	    "DB_Alarme".MLD[18].%X0 := "Ventil_Stati_DB".Mld."SF_CM05.QM61";
	    "DB_Alarme".MLD[18].%X1 := "Ventil_Stati_DB".Mld."TO_auf_CM05.QM64";
	    "DB_Alarme".MLD[18].%X2 := "Ventil_Stati_DB".Mld."TO_zu_CM05.QM64";
	    "DB_Alarme".MLD[18].%X3 := "Ventil_Stati_DB".Mld."SF_CM05.QM64";
	    "DB_Alarme".MLD[18].%X4 := "Ventil_Stati_DB".Mld."TO_auf_GP01.QM15";
	    "DB_Alarme".MLD[18].%X5 := "Ventil_Stati_DB".Mld."TO_zu_GP01.QM15";
	    "DB_Alarme".MLD[18].%X6 := "Ventil_Stati_DB".Mld."SF_GP01.QM15";
	    "DB_Alarme".MLD[18].%X7 := "Ventil_Stati_DB".Mld."TO_auf_GP01.QM16";
	    "DB_Alarme".MLD[18].%X8 := "Ventil_Stati_DB".Mld."TO_zu_GP01.QM16";
	    "DB_Alarme".MLD[18].%X9 := "Ventil_Stati_DB".Mld."SF_GP01.QM16";
	    "DB_Alarme".MLD[18].%X10 := "Ventil_Stati_DB".Mld."TO_auf_GP01.QM17";
	    "DB_Alarme".MLD[18].%X11 := "Ventil_Stati_DB".Mld."TO_zu_GP01.QM17";
	    "DB_Alarme".MLD[18].%X12 := "Ventil_Stati_DB".Mld."SF_GP01.QM17";
	    "DB_Alarme".MLD[18].%X13 := "Ventil_Stati_DB".Mld."TO_auf_GP01.QM18";
	    "DB_Alarme".MLD[18].%X14 := "Ventil_Stati_DB".Mld."TO_zu_GP01.QM18";
	    "DB_Alarme".MLD[18].%X15 := "Ventil_Stati_DB".Mld."SF_GP01.QM18";
	    
	    "DB_Alarme".MLD[19].%X0 := "Ventil_Stati_DB".Mld."TO_auf_GP01.QM19";
	    "DB_Alarme".MLD[19].%X1 := "Ventil_Stati_DB".Mld."TO_zu_GP01.QM19";
	    "DB_Alarme".MLD[19].%X2 := "Ventil_Stati_DB".Mld."SF_GP01.QM19";
	    "DB_Alarme".MLD[19].%X3 := "Ventil_Stati_DB".Mld."TO_auf_GP01.QM20";
	    "DB_Alarme".MLD[19].%X4 := "Ventil_Stati_DB".Mld."TO_zu_GP01.QM20";
	    "DB_Alarme".MLD[19].%X5 := "Ventil_Stati_DB".Mld."SF_GP01.QM20";
	    "DB_Alarme".MLD[19].%X6 := "Ventil_Stati_DB".Mld."TO_auf_GP01.QM21";
	    "DB_Alarme".MLD[19].%X7 := "Ventil_Stati_DB".Mld."TO_zu_GP01.QM21";
	    "DB_Alarme".MLD[19].%X8 := "Ventil_Stati_DB".Mld."SF_GP01.QM21";
	    "DB_Alarme".MLD[19].%X9 := "Ventil_Stati_DB".Mld."TO_auf_GP01.QM22";
	    "DB_Alarme".MLD[19].%X10 := "Ventil_Stati_DB".Mld."TO_zu_GP01.QM22";
	    "DB_Alarme".MLD[19].%X11 := "Ventil_Stati_DB".Mld."SF_GP01.QM22";
	    "DB_Alarme".MLD[19].%X12 := "Ventil_Stati_DB".Mld."TO_auf_GP02.QM38";
	    "DB_Alarme".MLD[19].%X13 := "Ventil_Stati_DB".Mld."TO_zu_GP02.QM38";
	    "DB_Alarme".MLD[19].%X14 := "Ventil_Stati_DB".Mld."SF_GP02.QM38";
	    "DB_Alarme".MLD[19].%X15 := "Ventil_Stati_DB".Mld."TO_auf_GP02.QM39";
	    
	    "DB_Alarme".MLD[20].%X0 := "Ventil_Stati_DB".Mld."TO_zu_GP02.QM39";
	    "DB_Alarme".MLD[20].%X1 := "Ventil_Stati_DB".Mld."SF_GP02.QM39";
	    "DB_Alarme".MLD[20].%X2 := "Ventil_Stati_DB".Mld."TO_auf_GP02.QM40";
	    "DB_Alarme".MLD[20].%X3 := "Ventil_Stati_DB".Mld."TO_zu_GP02.QM40";
	    "DB_Alarme".MLD[20].%X4 := "Ventil_Stati_DB".Mld."SF_GP02.QM40";
	    "DB_Alarme".MLD[20].%X5 := "Ventil_Stati_DB".Mld."TO_auf_GP02.QM41";
	    "DB_Alarme".MLD[20].%X6 := "Ventil_Stati_DB".Mld."TO_zu_GP02.QM41";
	    "DB_Alarme".MLD[20].%X7 := "Ventil_Stati_DB".Mld."SF_GP02.QM41";
	    "DB_Alarme".MLD[20].%X8 := "Ventil_Stati_DB".Mld."TO_auf_GP02.QM42";
	    "DB_Alarme".MLD[20].%X9 := "Ventil_Stati_DB".Mld."TO_zu_GP02.QM42";
	    "DB_Alarme".MLD[20].%X10 := "Ventil_Stati_DB".Mld."SF_GP02.QM42";
	    "DB_Alarme".MLD[20].%X11 := "Ventil_Stati_DB".Mld."TO_auf_GP02.QM43";
	    "DB_Alarme".MLD[20].%X12 := "Ventil_Stati_DB".Mld."TO_zu_GP02.QM43";
	    "DB_Alarme".MLD[20].%X13 := "Ventil_Stati_DB".Mld."SF_GP02.QM43";
	    "DB_Alarme".MLD[20].%X14 := "Ventil_Stati_DB".Mld."TO_auf_GP02.QM44";
	    "DB_Alarme".MLD[20].%X15 := "Ventil_Stati_DB".Mld."TO_zu_GP02.QM44";
	    
	    "DB_Alarme".MLD[21].%X0 := "Ventil_Stati_DB".Mld."SF_GP02.QM44";
	    "DB_Alarme".MLD[21].%X1 := "Ventil_Stati_DB".Mld."TO_auf_GP02.QM45";
	    "DB_Alarme".MLD[21].%X2 := "Ventil_Stati_DB".Mld."TO_zu_GP02.QM45";
	    "DB_Alarme".MLD[21].%X3 := "Ventil_Stati_DB".Mld."SF_GP02.QM45";
	    "DB_Alarme".MLD[21].%X4 := "Ventil_Stati_DB".Mld."TO_auf_GP02.QM46";
	    "DB_Alarme".MLD[21].%X5 := "Ventil_Stati_DB".Mld."TO_zu_GP02.QM46";
	    "DB_Alarme".MLD[21].%X6 := "Ventil_Stati_DB".Mld."SF_GP02.QM46";
	    "DB_Alarme".MLD[21].%X7 := "Ventil_Stati_DB".Mld."TO_auf_GP01.QM14";
	    "DB_Alarme".MLD[21].%X8 := "Ventil_Stati_DB".Mld."TO_zu_GP01.QM14";
	    "DB_Alarme".MLD[21].%X9 := "Ventil_Stati_DB".Mld."SF_GP01.QM14";
	    "DB_Alarme".MLD[21].%X10 := "FP_CM01.GP01".Mld.Drucktest_Filter_ok;
	    "DB_Alarme".MLD[21].%X11 := "FP_CM01.GP01".Mld.Drucktest_Filter_Fehler;
	    "DB_Alarme".MLD[21].%X12 := "FP_CM02.GP04".Mld.Drucktest_Filter_ok;
	    "DB_Alarme".MLD[21].%X13 := "FP_CM02.GP04".Mld.Drucktest_Filter_Fehler;
	    "DB_Alarme".MLD[21].%X14 := "FP_CM01.GP01".Mld.Drucktest_Filter_erfordert;
	    "DB_Alarme".MLD[21].%X15 := "FP_CM02.GP04".Mld.Drucktest_Filter_erfordert;
	    
	    "DB_Alarme".MLD[22].%X0 := "DI_FW_1".MLD.Alarm_HW.PosSys;
	    "DB_Alarme".MLD[22].%X1 := "DI_FW_1".MLD.Alarm_HW.BE_rck;
	    "DB_Alarme".MLD[22].%X2 := "DI_FW_1".MLD.Alarm_HW.BE_vor;
	    "DB_Alarme".MLD[22].%X3 := "DI_FW_1".MLD.Alarm_HW.HubSys_li;
	    "DB_Alarme".MLD[22].%X4 := "DI_FW_1".MLD.Alarm_HW.HubSys_re;
	    "DB_Alarme".MLD[22].%X5 := "DI_FW_1".MLD.Alarm_HW.GE_oben_li;
	    "DB_Alarme".MLD[22].%X6 := "DI_FW_1".MLD.Alarm_HW.GE_unten_li;
	    "DB_Alarme".MLD[22].%X7 := "DI_FW_1".MLD.Alarm_HW.GE_oben_re;
	    "DB_Alarme".MLD[22].%X8 := "DI_FW_1".MLD.Alarm_HW.GE_unten_re;
	    "DB_Alarme".MLD[22].%X9 := "DI_FW_1".MLD.Alarm_HW.Koll_LF;
	    "DB_Alarme".MLD[22].%X10 := "DI_FW_1".MLD.Alarm_HW.Koll_WF;
	    "DB_Alarme".MLD[22].%X11 := "DI_FW_1".MLD.Alarm_HW.Afs_BS;
	    "DB_Alarme".MLD[22].%X12 := "DI_FW_1".MLD.Alarm_HW.Afs_WS;
	    "DB_Alarme".MLD[22].%X13 := "DI_FW_1".MLD.Alarm_HW.GurtUeL_li;
	    "DB_Alarme".MLD[22].%X14 := "DI_FW_1".MLD.Alarm_HW.GurtUeL_re;
	    "DB_Alarme".MLD[22].%X15 := "DI_FW_1".MLD.Alarm_HW.St_FU_Fahrt;
	    
	    "DB_Alarme".MLD[23].%X0 := "DI_FW_1".MLD.Alarm_HW.F_Brk_Hub_li;
	    "DB_Alarme".MLD[23].%X1 := "DI_FW_1".MLD.Alarm_HW.F_Brk_Hub_re;
	    "DB_Alarme".MLD[23].%X2 := "DI_FW_1".MLD.Alarm_HW.F_Brk_Fahr;
	    "DB_Alarme".MLD[23].%X3 := "DI_FW_1".MLD.Alarm_HW.St_FU_Hub_li;
	    "DB_Alarme".MLD[23].%X4 := "DI_FW_1".MLD.Alarm_HW.St_FU_Hub_re;
	    "DB_Alarme".MLD[23].%X5 := "DI_FW_1".MLD.Alarm_HW.Last_UeW_li;
	    "DB_Alarme".MLD[23].%X6 := "DI_FW_1".MLD.Alarm_HW.Last_UeW_re;
	    "DB_Alarme".MLD[23].%X7 := "DI_FW_1".MLD.Alarm_HW.Temp_Fahrt;
	    "DB_Alarme".MLD[23].%X8 := "DI_FW_1".MLD.Alarm_HW.Temp_Hub;
	    "DB_Alarme".MLD[23].%X9 := "DI_FW_1".MLD.Alarm_HW.Laser_TF;
	    "DB_Alarme".MLD[23].%X10 := "DI_FW_1".MLD.Alarm_HW.Laser_PL;
	    "DB_Alarme".MLD[23].%X11 := "DI_FW_1".MLD.Alarm_HW.Profinet_nok;
	    "DB_Alarme".MLD[23].%X12 := "DI_FW_1".MLD.Alarm_HW.res_1;
	    "DB_Alarme".MLD[23].%X13 := "DI_FW_1".MLD.Alarm_HW.res_2;
	    "DB_Alarme".MLD[23].%X14 := "DI_FW_1".MLD.Alarm_HW.res_3;
	    "DB_Alarme".MLD[23].%X15 := "DI_FW_1".MLD.Alarm_HW.res_4;
	    
	    "DB_Alarme".MLD[24].%X0 := "DI_FW_1".MLD.Alarm_SW.Fehler_Quitt;
	    "DB_Alarme".MLD[24].%X1 := "DI_FW_1".MLD.Alarm_SW.BA_ungueltig;
	    "DB_Alarme".MLD[24].%X2 := "DI_FW_1".MLD.Alarm_SW.ProgErr;
	    "DB_Alarme".MLD[24].%X3 := "DI_FW_1".MLD.Alarm_SW.nReferenz;
	    "DB_Alarme".MLD[24].%X4 := "DI_FW_1".MLD.Alarm_SW.NotStop;
	    "DB_Alarme".MLD[24].%X5 := "DI_FW_1".MLD.Alarm_SW.Laser_off;
	    "DB_Alarme".MLD[24].%X6 := "DI_FW_1".MLD.Alarm_SW.TO_Fahrt;
	    "DB_Alarme".MLD[24].%X7 := "DI_FW_1".MLD.Alarm_SW.Auto_SU;
	    "DB_Alarme".MLD[24].%X8 := "DI_FW_1".MLD.Alarm_SW.Auto_WT;
	    "DB_Alarme".MLD[24].%X9 := "DI_FW_1".MLD.Alarm_SW.WT_change;
	    "DB_Alarme".MLD[24].%X10 := "DI_FW_1".MLD.Alarm_SW.Hub_not_mittig_li;
	    "DB_Alarme".MLD[24].%X11 := "DI_FW_1".MLD.Alarm_SW.Hub_nen_li;
	    "DB_Alarme".MLD[24].%X12 := "DI_FW_1".MLD.Alarm_SW.TO_Hub_li;
	    "DB_Alarme".MLD[24].%X13 := "DI_FW_1".MLD.Alarm_SW.Senken_WT_li;
	    "DB_Alarme".MLD[24].%X14 := "DI_FW_1".MLD.Alarm_SW.Senken_Sperre_li;
	    "DB_Alarme".MLD[24].%X15 := "DI_FW_1".MLD.Alarm_SW.Heben_WT_li;
	    
	    "DB_Alarme".MLD[25].%X0 := "DI_FW_1".MLD.Alarm_SW.SO_fehlt_li;
	    "DB_Alarme".MLD[25].%X1 := "DI_FW_1".MLD.Alarm_SW.SU_fehlt_li;
	    "DB_Alarme".MLD[25].%X2 := "DI_FW_1".MLD.Alarm_SW.PosTyp_WT_Typ_li;
	    "DB_Alarme".MLD[25].%X3 := "DI_FW_1".MLD.Alarm_SW.WTon_bei_SU_li;
	    "DB_Alarme".MLD[25].%X4 := "DI_FW_1".MLD.Alarm_SW.TO_Hub_re;
	    "DB_Alarme".MLD[25].%X5 := "DI_FW_1".MLD.Alarm_SW.Senken_WT_re;
	    "DB_Alarme".MLD[25].%X6 := "DI_FW_1".MLD.Alarm_SW.Senken_Sperre_re;
	    "DB_Alarme".MLD[25].%X7 := "DI_FW_1".MLD.Alarm_SW.Heben_WT_re;
	    "DB_Alarme".MLD[25].%X8 := "DI_FW_1".MLD.Alarm_SW.SO_fehlt_re;
	    "DB_Alarme".MLD[25].%X9 := "DI_FW_1".MLD.Alarm_SW.SU_fehlt_re;
	    "DB_Alarme".MLD[25].%X10 := "DI_FW_1".MLD.Alarm_SW.PosTyp_WT_Typ_re;
	    "DB_Alarme".MLD[25].%X11 := "DI_FW_1".MLD.Alarm_SW.WTon_bei_SU_re;
	    "DB_Alarme".MLD[25].%X12 := "DI_FW_1".MLD.Alarm_SW.Hub_not_mittig_re;
	    "DB_Alarme".MLD[25].%X13 := "DI_FW_1".MLD.Alarm_SW.Hub_nen_re;
	    "DB_Alarme".MLD[25].%X14 := "DI_FW_1".MLD.Alarm_SW.ALSW_31;
	    "DB_Alarme".MLD[25].%X15 := "DI_FW_1".MLD.Alarm_SW.TO_Befehl;
	    
	    "DB_Alarme".MLD[26].%X0 := "DI_FW_1".MLD.Warnung.Optik_PosSys;
	    "DB_Alarme".MLD[26].%X1 := "DI_FW_1".MLD.Warnung.Temp_PosSys;
	    "DB_Alarme".MLD[26].%X2 := "DI_FW_1".MLD.Warnung.Temp_Fahrt;
	    "DB_Alarme".MLD[26].%X3 := "DI_FW_1".MLD.Warnung.Temp_Hub;
	    "DB_Alarme".MLD[26].%X4 := "DI_FW_1".MLD.Warnung.LSA;
	    "DB_Alarme".MLD[26].%X5 := "DI_FW_1".MLD.Warnung.Bh0;
	    "DB_Alarme".MLD[26].%X6 := "DI_FW_1".MLD.Warnung.Bh100;
	    "DB_Alarme".MLD[26].%X7 := "DI_FW_1".MLD.Warnung.Bh1000;
	    "DB_Alarme".MLD[26].%X8 := "DI_FW_1".MLD.Warnung.Wrn_Plaus_PosSys;
	    "DB_Alarme".MLD[26].%X9 := "DI_FW_1".MLD.Warnung.Wrn_WZ_niO_li_1;
	    "DB_Alarme".MLD[26].%X10 := "DI_FW_1".MLD.Warnung.Wrn_WZ_niO_li_2;
	    "DB_Alarme".MLD[26].%X11 := "DI_FW_1".MLD.Warnung.Wrn_WZ_niO_li_3;
	    "DB_Alarme".MLD[26].%X12 := "DI_FW_1".MLD.Warnung.Wrn_WZ_niO_li_4;
	    "DB_Alarme".MLD[26].%X13 := "DI_FW_1".MLD.Warnung.Wrn_WZ_niO_re_1;
	    "DB_Alarme".MLD[26].%X14 := "DI_FW_1".MLD.Warnung.Wrn_WZ_niO_re_2;
	    "DB_Alarme".MLD[26].%X15 := "DI_FW_1".MLD.Warnung.Wrn_WZ_niO_re_3;
	    
	    "DB_Alarme".MLD[27].%X0 := "DI_FW_1".MLD.Warnung.Wrn_WZ_niO_re_4;
	    "DB_Alarme".MLD[27].%X1 := "DI_FW_1".MLD.Warnung.WARN_18;
	    "DB_Alarme".MLD[27].%X2 := "DI_FW_1".MLD.Warnung.WARN_19;
	    "DB_Alarme".MLD[27].%X3 := "DI_FW_1".MLD.Warnung.WARN_20;
	    "DB_Alarme".MLD[27].%X4 := "DI_FW_1".MLD.Warnung.WARN_21;
	    "DB_Alarme".MLD[27].%X5 := "DI_FW_1".MLD.Warnung.WARN_22;
	    "DB_Alarme".MLD[27].%X6 := "DI_FW_1".MLD.Warnung.WARN_23;
	    "DB_Alarme".MLD[27].%X7 := "DI_FW_1".MLD.Warnung.WARN_24;
	    "DB_Alarme".MLD[27].%X8 := "DI_FW_1".MLD.Warnung.WARN_25;
	    "DB_Alarme".MLD[27].%X9 := "DI_FW_1".MLD.Warnung.WARN_26;
	    "DB_Alarme".MLD[27].%X10 := "DI_FW_1".MLD.Warnung.WARN_27;
	    "DB_Alarme".MLD[27].%X11 := "DI_FW_1".MLD.Warnung.WARN_28;
	    "DB_Alarme".MLD[27].%X12 := "DI_FW_1".MLD.Warnung.WARN_29;
	    "DB_Alarme".MLD[27].%X13 := "DI_FW_1".MLD.Warnung.WARN_30;
	    "DB_Alarme".MLD[27].%X14 := "DI_FW_1".MLD.Warnung.WARN_WT_nUms;
	    "DB_Alarme".MLD[27].%X15 := "DI_FW_1".MLD.Warnung.WARN_nAuto;
	    
	    "DB_Alarme".MLD[28].%X0 := "DI_QF_WR02_03".Mld.TO_WR02;
	    "DB_Alarme".MLD[28].%X1 := "DI_QF_WR02_03".Mld.TO_WR03;
	    "DB_Alarme".MLD[28].%X2 := "DI_QF_WR02_03".Mld.St_FU_WR02;
	    "DB_Alarme".MLD[28].%X3 := "DI_QF_WR02_03".Mld.St_FU_WR03;
	    "DB_Alarme".MLD[28].%X4 := "DI_QF_WR02_03".Mld.FU_nichtbereit_WR02;
	    "DB_Alarme".MLD[28].%X5 := "DI_QF_WR02_03".Mld.FU_nichtbereit_WR03;
	    "DB_Alarme".MLD[28].%X6 := "DI_QF_WR02_03".Mld.SF_WR02;
	    "DB_Alarme".MLD[28].%X7 := "DI_QF_WR02_03".Mld.SF_WR03;
	    "DB_Alarme".MLD[28].%X8 := FALSE;
	    "DB_Alarme".MLD[28].%X9 := "FP_CM01.GP01".Mld.Pu_Spuelen_Fertig;
	    "DB_Alarme".MLD[28].%X10 := "FP_CM02.GP04".Mld.Pu_Spuelen_Fertig;
	    "DB_Alarme".MLD[28].%X11 := "UP_CM01.GP02".Mld.Pu_Spuelen_Fertig;
	    "DB_Alarme".MLD[28].%X12 := "UP_CM02.GP05".Mld.Pu_Spuelen_Fertig;
	    "DB_Alarme".MLD[28].%X13 := "UP_CM03.GP03".Mld.Pu_Spuelen_Fertig;
	    "DB_Alarme".MLD[28].%X14 := "UP_CM04.GP06".Mld.Pu_Spuelen_Fertig;
	    "DB_Alarme".MLD[28].%X15 := "Pu_CM05.GP11_DB".Mld.Pu_Spuelen_Fertig;
	    
	    "DB_Alarme".MLD[29].%X0 := "DB_Korbumlaeufe".Korb[1].Warnung;
	    "DB_Alarme".MLD[29].%X1 := "DB_Korbumlaeufe".Korb[1].max_erreicht;
	    "DB_Alarme".MLD[29].%X2 := "DB_Korbumlaeufe".Korb[2].Warnung;
	    "DB_Alarme".MLD[29].%X3 := "DB_Korbumlaeufe".Korb[2].max_erreicht;
	    "DB_Alarme".MLD[29].%X4 := "DB_Korbumlaeufe".Korb[3].Warnung;
	    "DB_Alarme".MLD[29].%X5 := "DB_Korbumlaeufe".Korb[3].max_erreicht;
	    "DB_Alarme".MLD[29].%X6 := "DB_Korbumlaeufe".Korb[4].Warnung;
	    "DB_Alarme".MLD[29].%X7 := "DB_Korbumlaeufe".Korb[4].max_erreicht;
	    "DB_Alarme".MLD[29].%X8 := "DB_Korbumlaeufe".Korb[5].Warnung;
	    "DB_Alarme".MLD[29].%X9 := "DB_Korbumlaeufe".Korb[5].max_erreicht;
	    "DB_Alarme".MLD[29].%X10 := "DB_Korbumlaeufe".Korb[6].Warnung;
	    "DB_Alarme".MLD[29].%X11 := "DB_Korbumlaeufe".Korb[6].max_erreicht;
	    "DB_Alarme".MLD[29].%X12 := "DB_Korbumlaeufe".Korb[7].Warnung;
	    "DB_Alarme".MLD[29].%X13 := "DB_Korbumlaeufe".Korb[7].max_erreicht;
	    "DB_Alarme".MLD[29].%X14 := "DB_Korbumlaeufe".Korb[8].Warnung;
	    "DB_Alarme".MLD[29].%X15 := "DB_Korbumlaeufe".Korb[8].max_erreicht;
	        
	    "DB_Alarme".MLD[30].%X0 := "DB_Korbumlaeufe".Korb[9].Warnung;
	    "DB_Alarme".MLD[30].%X1 := "DB_Korbumlaeufe".Korb[9].max_erreicht;
	    "DB_Alarme".MLD[30].%X2 := "DB_Korbumlaeufe".Korb[10].Warnung;
	    "DB_Alarme".MLD[30].%X3 := "DB_Korbumlaeufe".Korb[10].max_erreicht;
	    "DB_Alarme".MLD[30].%X4 := "DB_Korbumlaeufe".Korb[11].Warnung;
	    "DB_Alarme".MLD[30].%X5 := "DB_Korbumlaeufe".Korb[11].max_erreicht;
	    "DB_Alarme".MLD[30].%X6 := "DB_Korbumlaeufe".Korb[12].Warnung;
	    "DB_Alarme".MLD[30].%X7 := "DB_Korbumlaeufe".Korb[12].max_erreicht;
	    "DB_Alarme".MLD[30].%X8 := "DB_Korbumlaeufe".Korb[13].Warnung;
	    "DB_Alarme".MLD[30].%X9 := "DB_Korbumlaeufe".Korb[13].max_erreicht;
	    "DB_Alarme".MLD[30].%X10 := "FP_CM01.GP01".Mld.Filterbeutel_Wechsel_Vorwarngrenze;
	    "DB_Alarme".MLD[30].%X11 := "FP_CM01.GP01".Mld.Filterbeutel_Wechsel_notwendig;
	    "DB_Alarme".MLD[30].%X12 := "FP_CM02.GP04".Mld.Filterbeutel_Wechsel_Vorwarngrenze;
	    "DB_Alarme".MLD[30].%X13 := "FP_CM02.GP04".Mld.Filterbeutel_Wechsel_notwendig;
	    "DB_Alarme".MLD[30].%X14 :=  "Pu_GP01.GP13".Mld.UeW_Dfl_Dos;
	    "DB_Alarme".MLD[30].%X15 := "Pu_GP02.GP10".Mld.UeW_Dfl_Dos;
	    
	    "DB_Alarme".MLD[31].%X0 := "FP_CM01.GP01".Mld.Drucktest_Pumpe_ok;
	    "DB_Alarme".MLD[31].%X1 := "FP_CM01.GP01".Mld.Drucktest_Pumpe_Fehler;
	    "DB_Alarme".MLD[31].%X2 := "FP_CM02.GP04".Mld.Drucktest_Pumpe_ok;
	    "DB_Alarme".MLD[31].%X3 := "FP_CM02.GP04".Mld.Drucktest_Pumpe_Fehler;
	    "DB_Alarme".MLD[31].%X4 := "UP_CM01.GP02".Mld.Drucktest_ok;
	    "DB_Alarme".MLD[31].%X5 := "UP_CM01.GP02".Mld.DT_Fehler;
	    "DB_Alarme".MLD[31].%X6 := "UP_CM02.GP05".Mld.Drucktest_ok;
	    "DB_Alarme".MLD[31].%X7 := "UP_CM02.GP05".Mld.DT_Fehler;
	    "DB_Alarme".MLD[31].%X8 := "UP_CM03.GP03".Mld.Drucktest_ok;
	    "DB_Alarme".MLD[31].%X9 := "UP_CM03.GP03".Mld.DT_Fehler;
	    "DB_Alarme".MLD[31].%X10 := "UP_CM04.GP06".Mld.Drucktest_ok;
	    "DB_Alarme".MLD[31].%X11 := "UP_CM04.GP06".Mld.DT_Fehler;
	    "DB_Alarme".MLD[31].%X12 := "Pu_CM05.GP11_DB".Mld.Drucktest_ok;
	    "DB_Alarme".MLD[31].%X13 := "Pu_CM05.GP11_DB".Mld.DT_Fehler;
	    "DB_Alarme".MLD[31].%X14 := "UP_CM01.GP02".Mld.UeW_Dfl_Ents;
	    "DB_Alarme".MLD[31].%X15 := "UP_CM02.GP05".Mld.UeW_Dfl_Ents;
	    
	        REGION Reserve
	        
	        "DB_Alarme".MLD[32].%X0 := FALSE;
	        "DB_Alarme".MLD[32].%X1 := FALSE;
	        "DB_Alarme".MLD[32].%X2 := FALSE;
	        "DB_Alarme".MLD[32].%X3 := FALSE;
	        "DB_Alarme".MLD[32].%X4 := FALSE;
	        "DB_Alarme".MLD[32].%X5 := FALSE;
	        "DB_Alarme".MLD[32].%X6 := FALSE;
	        "DB_Alarme".MLD[32].%X7 := FALSE;
	        "DB_Alarme".MLD[32].%X8 := FALSE;
	        "DB_Alarme".MLD[32].%X9 := FALSE;
	        "DB_Alarme".MLD[32].%X10 := FALSE;
	        "DB_Alarme".MLD[32].%X11 := FALSE;
	        "DB_Alarme".MLD[32].%X12 := FALSE;
	        "DB_Alarme".MLD[32].%X13 := FALSE;
	        "DB_Alarme".MLD[32].%X14 := FALSE;
	        "DB_Alarme".MLD[32].%X15 := FALSE;
	        
	        "DB_Alarme".MLD[33].%X0 := FALSE;
	        "DB_Alarme".MLD[33].%X1 := FALSE;
	        "DB_Alarme".MLD[33].%X2 := FALSE;
	        "DB_Alarme".MLD[33].%X3 := FALSE;
	        "DB_Alarme".MLD[33].%X4 := FALSE;
	        "DB_Alarme".MLD[33].%X5 := FALSE;
	        "DB_Alarme".MLD[33].%X6 := FALSE;
	        "DB_Alarme".MLD[33].%X7 := FALSE;
	        "DB_Alarme".MLD[33].%X8 := FALSE;
	        "DB_Alarme".MLD[33].%X9 := FALSE;
	        "DB_Alarme".MLD[33].%X10 := FALSE;
	        "DB_Alarme".MLD[33].%X11 := FALSE;
	        "DB_Alarme".MLD[33].%X12 := FALSE;
	        "DB_Alarme".MLD[33].%X13 := FALSE;
	        "DB_Alarme".MLD[33].%X14 := FALSE;
	        "DB_Alarme".MLD[33].%X15 := FALSE;
	        
	        "DB_Alarme".MLD[34].%X0 := FALSE;
	        "DB_Alarme".MLD[34].%X1 := FALSE;
	        "DB_Alarme".MLD[34].%X2 := FALSE;
	        "DB_Alarme".MLD[34].%X3 := FALSE;
	        "DB_Alarme".MLD[34].%X4 := FALSE;
	        "DB_Alarme".MLD[34].%X5 := FALSE;
	        "DB_Alarme".MLD[34].%X6 := FALSE;
	        "DB_Alarme".MLD[34].%X7 := FALSE;
	        "DB_Alarme".MLD[34].%X8 := FALSE;
	        "DB_Alarme".MLD[34].%X9 := FALSE;
	        "DB_Alarme".MLD[34].%X10 := FALSE;
	        "DB_Alarme".MLD[34].%X11 := FALSE;
	        "DB_Alarme".MLD[34].%X12 := FALSE;
	        "DB_Alarme".MLD[34].%X13 := FALSE;
	        "DB_Alarme".MLD[34].%X14 := FALSE;
	        "DB_Alarme".MLD[34].%X15 := FALSE;
	        
	        "DB_Alarme".MLD[35].%X0 := FALSE;
	        "DB_Alarme".MLD[35].%X1 := FALSE;
	        "DB_Alarme".MLD[35].%X2 := FALSE;
	        "DB_Alarme".MLD[35].%X3 := FALSE;
	        "DB_Alarme".MLD[35].%X4 := FALSE;
	        "DB_Alarme".MLD[35].%X5 := FALSE;
	        "DB_Alarme".MLD[35].%X6 := FALSE;
	        "DB_Alarme".MLD[35].%X7 := FALSE;
	        "DB_Alarme".MLD[35].%X8 := FALSE;
	        "DB_Alarme".MLD[35].%X9 := FALSE;
	        "DB_Alarme".MLD[35].%X10 := FALSE;
	        "DB_Alarme".MLD[35].%X11 := FALSE;
	        "DB_Alarme".MLD[35].%X12 := FALSE;
	        "DB_Alarme".MLD[35].%X13 := FALSE;
	        "DB_Alarme".MLD[35].%X14 := FALSE;
	        "DB_Alarme".MLD[35].%X15 := FALSE;
	        
	        "DB_Alarme".MLD[36].%X0 := FALSE;
	        "DB_Alarme".MLD[36].%X1 := FALSE;
	        "DB_Alarme".MLD[36].%X2 := FALSE;
	        "DB_Alarme".MLD[36].%X3 := FALSE;
	        "DB_Alarme".MLD[36].%X4 := FALSE;
	        "DB_Alarme".MLD[36].%X5 := FALSE;
	        "DB_Alarme".MLD[36].%X6 := FALSE;
	        "DB_Alarme".MLD[36].%X7 := FALSE;
	        "DB_Alarme".MLD[36].%X8 := FALSE;
	        "DB_Alarme".MLD[36].%X9 := FALSE;
	        "DB_Alarme".MLD[36].%X10 := FALSE;
	        "DB_Alarme".MLD[36].%X11 := FALSE;
	        "DB_Alarme".MLD[36].%X12 := FALSE;
	        "DB_Alarme".MLD[36].%X13 := FALSE;
	        "DB_Alarme".MLD[36].%X14 := FALSE;
	        "DB_Alarme".MLD[36].%X15 := FALSE;
	        
	        "DB_Alarme".MLD[37].%X0 := FALSE;
	        "DB_Alarme".MLD[37].%X1 := FALSE;
	        "DB_Alarme".MLD[37].%X2 := FALSE;
	        "DB_Alarme".MLD[37].%X3 := FALSE;
	        "DB_Alarme".MLD[37].%X4 := FALSE;
	        "DB_Alarme".MLD[37].%X5 := FALSE;
	        "DB_Alarme".MLD[37].%X6 := FALSE;
	        "DB_Alarme".MLD[37].%X7 := FALSE;
	        "DB_Alarme".MLD[37].%X8 := FALSE;
	        "DB_Alarme".MLD[37].%X9 := FALSE;
	        "DB_Alarme".MLD[37].%X10 := FALSE;
	        "DB_Alarme".MLD[37].%X11 := FALSE;
	        "DB_Alarme".MLD[37].%X12 := FALSE;
	        "DB_Alarme".MLD[37].%X13 := FALSE;
	        "DB_Alarme".MLD[37].%X14 := FALSE;
	        "DB_Alarme".MLD[37].%X15 := FALSE;
	        
	        "DB_Alarme".MLD[38].%X0 := FALSE;
	        "DB_Alarme".MLD[38].%X1 := FALSE;
	        "DB_Alarme".MLD[38].%X2 := FALSE;
	        "DB_Alarme".MLD[38].%X3 := FALSE;
	        "DB_Alarme".MLD[38].%X4 := FALSE;
	        "DB_Alarme".MLD[38].%X5 := FALSE;
	        "DB_Alarme".MLD[38].%X6 := FALSE;
	        "DB_Alarme".MLD[38].%X7 := FALSE;
	        "DB_Alarme".MLD[38].%X8 := FALSE;
	        "DB_Alarme".MLD[38].%X9 := FALSE;
	        "DB_Alarme".MLD[38].%X10 := FALSE;
	        "DB_Alarme".MLD[38].%X11 := FALSE;
	        "DB_Alarme".MLD[38].%X12 := FALSE;
	        "DB_Alarme".MLD[38].%X13 := FALSE;
	        "DB_Alarme".MLD[38].%X14 := FALSE;
	        "DB_Alarme".MLD[38].%X15 := FALSE;
	        
	        "DB_Alarme".MLD[39].%X0 := FALSE;
	        "DB_Alarme".MLD[39].%X1 := FALSE;
	        "DB_Alarme".MLD[39].%X2 := FALSE;
	        "DB_Alarme".MLD[39].%X3 := FALSE;
	        "DB_Alarme".MLD[39].%X4 := FALSE;
	        "DB_Alarme".MLD[39].%X5 := FALSE;
	        "DB_Alarme".MLD[39].%X6 := FALSE;
	        "DB_Alarme".MLD[39].%X7 := FALSE;
	        "DB_Alarme".MLD[39].%X8 := FALSE;
	        "DB_Alarme".MLD[39].%X9 := FALSE;
	        "DB_Alarme".MLD[39].%X10 := FALSE;
	        "DB_Alarme".MLD[39].%X11 := FALSE;
	        "DB_Alarme".MLD[39].%X12 := FALSE;
	        "DB_Alarme".MLD[39].%X13 := FALSE;
	        "DB_Alarme".MLD[39].%X14 := FALSE;
	        "DB_Alarme".MLD[39].%X15 := FALSE;
	        
	        "DB_Alarme".MLD[40].%X0 := FALSE;
	        "DB_Alarme".MLD[40].%X1 := FALSE;
	        "DB_Alarme".MLD[40].%X2 := FALSE;
	        "DB_Alarme".MLD[40].%X3 := FALSE;
	        "DB_Alarme".MLD[40].%X4 := FALSE;
	        "DB_Alarme".MLD[40].%X5 := FALSE;
	        "DB_Alarme".MLD[40].%X6 := FALSE;
	        "DB_Alarme".MLD[40].%X7 := FALSE;
	        "DB_Alarme".MLD[40].%X8 := FALSE;
	        "DB_Alarme".MLD[40].%X9 := FALSE;
	        "DB_Alarme".MLD[40].%X10 := FALSE;
	        "DB_Alarme".MLD[40].%X11 := FALSE;
	        "DB_Alarme".MLD[40].%X12 := FALSE;
	        "DB_Alarme".MLD[40].%X13 := FALSE;
	        "DB_Alarme".MLD[40].%X14 := FALSE;
	        "DB_Alarme".MLD[40].%X15 := FALSE;
	    END_REGION ;
	    
	END_REGION
	
	"FC_Mld_Leuchte_Hupe"(Max_Word := "Anzahl_Alarm_Woerter",
	                      La_Rot => #La_Rot,
	                      La_Gelb => #La_Gelb,
	                      La_Blau => #La_Blau);
	
	REGION Hupe
	    
	    //Quittung Hupe Rot
	    "DB_Alarme".Timer_Hupe_Rot.TON(IN := NOT "DB_Alarme".M_Q_Hupe_Rot AND NOT "DB_Alarme".Hupe_Dauer_Rot,
	    PT := "DB_Alarme".Zeit_Auto_Quitt_Hupe_Rot,
	    Q => #Hupe_Quitt_Rot);
	    
	    IF "DB_Alarme".IN_Quitt_Hupe OR #Hupe_Quitt_Rot THEN
	        "DB_Alarme".M_Q_Hupe_Rot := true;
	        "DB_Alarme".Hupe_Dauer_Rot := FALSE;
	    END_IF;
	    
	    //Quittung Hupe Gelb
	    "DB_Alarme".Timer_Hupe_Gelb.TON(IN := NOT "DB_Alarme".M_Q_Hupe_Gelb AND NOT "DB_Alarme".Hupe_Dauer_Gelb,
	    PT := "DB_Alarme".Zeit_Auto_Quitt_Hupe_Gelb,
	    Q => #Hupe_Quitt_Gelb);
	    
	    IF "DB_Alarme".IN_Quitt_Hupe OR #Hupe_Quitt_Gelb THEN
	        "DB_Alarme".M_Q_Hupe_Gelb := true;
	        "DB_Alarme".Hupe_Dauer_Gelb := FALSE;
	    END_IF;
	    
	    //Quittung Hupe Blau
	    "DB_Alarme".Timer_Hupe_Blau.TON(IN := NOT "DB_Alarme".M_Q_Hupe_Blau AND NOT "DB_Alarme".Hupe_Dauer_Blau,
	    PT := "DB_Alarme".Zeit_Auto_Quitt_Hupe_Blau,
	    Q => #Hupe_Quitt_Blau);
	    
	    IF "DB_Alarme".IN_Quitt_Hupe OR #Hupe_Quitt_Blau  THEN
	        "DB_Alarme".M_Q_Hupe_Blau := true;
	        "DB_Alarme".Hupe_Dauer_Blau := FALSE;
	    END_IF;
	    
	    //Ausgänge beschreiben
	    "DB_ANLAGE".OUT.Stoerung_Aku  := NOT "DB_Alarme".M_Q_Hupe_Rot;
	    "DB_Alarme".Lampe_Rot := #La_Rot;
	    "DB_Alarme".Lampe_Gelb := #La_Gelb;
	    "DB_Alarme".Lampe_Blau := #La_Blau;
	    
	    "DB_ANLAGE".OUT.Fehler_Quitt := "DI_FW_1".ZST.FEHLER OR NOT "DB_PNOZ_Comm".connection.activate
	    OR "Deckel_CM01".Zst.Fehler OR "Deckel_CM02".Zst.Fehler OR "Tor".Zst.Fehler
	    OR "DI_QF_WR02_03".Zst.Fehler OR "DB_Alarme".La_Quit_Err;
	    
	END_REGION
	
END_FUNCTION

FUNCTION "FC_Mld_Leuchte_Hupe" : Void
{ S7_Optimized_Access := 'TRUE' }
VERSION : 0.1
   VAR_INPUT 
      Max_Word : Int;   // Anzahl Worte insgesamt
   END_VAR

   VAR_OUTPUT 
      La_Rot : Bool;
      La_Gelb : Bool;
      La_Blau : Bool;
   END_VAR

   VAR_TEMP 
      i : Int;
      j : Int;
      Temp_Mld : Array[0..15] of Bool;   // Inhalt eines Meldewortes
      Temp_AM_Mld : Array[0..15] of Bool;   // Inhalt des Altmerkerwortes
      Edit_Mld_change : Bool;
   END_VAR


BEGIN
	REGION Parameter
	    //für Editierfunktion in Visu
	    //Meldenummer fängt in Visu bei 1 an, daher -1 für Wort und Bitberechnung
	    
	    //Adressberechnung
	    "DB_Alarme".Edit.Edit_Meldewort := ("DB_Alarme".Edit.Edit_Meld - 1) / 16; //welches Meldewort
	    "DB_Alarme".Edit.Edit_Meldebit := ("DB_Alarme".Edit.Edit_Meld - 1) MOD 16; //welches Meldebit
	    
	    //Änderung der ausgewählten Meldung in Visu erkannt
	    "FC_Flanke"(In:="DB_Alarme".Edit.Edit_Meld <> "DB_Alarme".Edit.Edit_Meld_old,
	                  neg:=FALSE,
	                  Flanke=>#Edit_Mld_change,
	                  AM:="DB_Alarme".Edit.AM_Edit);
	    
	    //Neue Daten in Editierstruktur
	    IF #Edit_Mld_change AND "DB_Alarme".Edit.Edit_Meld <> 0 THEN
	        "DB_Alarme".Edit.Par := "DB_Alarme".Para_Mld["DB_Alarme".Edit.Edit_Meldewort].Parameter["DB_Alarme".Edit.Edit_Meldebit];
	        
	        "DB_Alarme".Edit.Edit_Meld_old := "DB_Alarme".Edit.Edit_Meld; //Altmerker
	        "DB_Alarme".Edit.Uebernommen := FALSE;
	    END_IF;
	    
	    //Daten übernehmen
	    IF "DB_Alarme".Edit.Uebernehmen THEN
	        "DB_Alarme".Para_Mld["DB_Alarme".Edit.Edit_Meldewort].Parameter["DB_Alarme".Edit.Edit_Meldebit] := "DB_Alarme".Edit.Par;
	        "DB_Alarme".Edit.Uebernommen := TRUE;
	        "DB_Alarme".Edit.Uebernehmen := FALSE;
	    END_IF;
	    
	    // Cancel changes
	    IF "DB_Alarme".Edit.Verwerfen THEN
	        "DB_Alarme".Edit.Par := "DB_Alarme".Para_Mld["DB_Alarme".Edit.Edit_Meldewort].Parameter["DB_Alarme".Edit.Edit_Meldebit];
	        "DB_Alarme".Edit.Verwerfen := FALSE;
	    END_IF;
	    
	    "DB_Alarme".Edit.Editiert := "FC_Alarm_Editiert_HMI"(IN1:="DB_Alarme".Para_Mld["DB_Alarme".Edit.Edit_Meldewort].Parameter["DB_Alarme".Edit.Edit_Meldebit], IN2:="DB_Alarme".Edit.Par);
	        
	END_REGION
	
	REGION Auswertung
	    //Parameterbyte:
	    //Hupe Rot und Lampe Rot sind Standard, alles andere wird übers Parabyte eingestellt
	    //generell Hupe automatisch Quittieren pro Meldung, wenn Dauerhupen gewünscht dann im Parabyte einstellen
	    
	    //Init Meldeleuchten und Hupenquittung
	    #La_Rot := FALSE;
	    #La_Gelb := FALSE;
	    #La_Blau := FALSE;
	    "DB_Alarme".La_Quit_Err := FALSE;
	    "DB_Alarme".auto_aus := FALSE;
	    "DB_Alarme".stop_request := FALSE;
	    
	    FOR #i := 0 TO #Max_Word DO
	        
	        SCATTER(IN := "DB_Alarme".MLD[#i], //Meldewort in Bitarray vereinzeln
	                OUT => #Temp_Mld);
	        SCATTER(IN := "DB_Alarme".AM_MLD[#i], //Altmerkerwort in Bitarray vereinzeln
	                OUT => #Temp_AM_Mld);
	        
	        //Meldewort bearbeiten
	        FOR #j := 0 TO 15 DO
	            
	            //Lampen und sonstige Bits
	            IF #Temp_Mld[#j] = TRUE THEN
	                IF "DB_Alarme".Para_Mld[#i].Parameter[#j].La_Gelb = TRUE THEN
	                    #La_Gelb := TRUE;
	                END_IF;
	                
	                IF "DB_Alarme".Para_Mld[#i].Parameter[#j].La_Blau = TRUE THEN
	                    #La_Blau := TRUE;
	                END_IF;
	                
	                IF "DB_Alarme".Para_Mld[#i].Parameter[#j].nicht_La_Rot = FALSE THEN
	                    #La_Rot := TRUE;
	                END_IF;
	                
	                IF "DB_Alarme".Para_Mld[#i].Parameter[#j].La_Quit_Err = TRUE THEN
	                    "DB_Alarme".La_Quit_Err := TRUE;
	                END_IF;
	                
	            END_IF;
	            
	            //Hupen
	            IF ((#Temp_Mld[#j] XOR #Temp_AM_Mld[#j]) AND #Temp_Mld[#j]) = TRUE THEN
	                IF "DB_Alarme".Para_Mld[#i].Parameter[#j].Hupe_Gelb = TRUE THEN
	                    "DB_Alarme".M_Q_Hupe_Gelb := false;
	                    IF "DB_Alarme".Para_Mld[#i].Parameter[#j].Hupe_Dauer_Gelb = TRUE THEN
	                        "DB_Alarme".Hupe_Dauer_Gelb := TRUE;
	                    END_IF;
	                END_IF;
	                
	                IF "DB_Alarme".Para_Mld[#i].Parameter[#j].Hupe_Blau = TRUE THEN
	                    "DB_Alarme".M_Q_Hupe_Blau := false;
	                    IF "DB_Alarme".Para_Mld[#i].Parameter[#j].Hupe_Dauer_Blau = TRUE THEN
	                        "DB_Alarme".Hupe_Dauer_Blau := TRUE;
	                    END_IF;
	                END_IF;
	                
	                IF "DB_Alarme".Para_Mld[#i].Parameter[#j].nicht_Hupe_Rot = FALSE THEN
	                    "DB_Alarme".M_Q_Hupe_Rot := false;
	                    IF "DB_Alarme".Para_Mld[#i].Parameter[#j].Hupe_Dauer_Rot = TRUE THEN
	                        "DB_Alarme".Hupe_Dauer_Rot := TRUE;
	                    END_IF;
	                END_IF;
	            END_IF;
	            
	        END_FOR;
	        
	        //auf Altmerker kopieren
	        "DB_Alarme".AM_MLD[#i] := "DB_Alarme".MLD[#i];
	        
	    END_FOR;
	    
	END_REGION
END_FUNCTION

FUNCTION "FC_Flanke" : Void
{ S7_Optimized_Access := 'TRUE' }
VERSION : 0.1
   VAR_INPUT 
      In : Bool;
      neg : Bool;
   END_VAR

   VAR_OUTPUT 
      Flanke : Bool;
   END_VAR

   VAR_IN_OUT 
      AM : Bool;
   END_VAR


BEGIN
	IF (#In = TRUE AND #AM = FALSE AND #neg = FALSE) OR (#In = FALSE AND #AM = TRUE AND #neg = TRUE) THEN
	    #Flanke := TRUE;
	ELSE
	    #Flanke := false;
	END_IF;
	
	#AM := #In;
	
END_FUNCTION

FUNCTION "FC_Alarm_Editiert_HMI" : Bool
{ S7_Optimized_Access := 'TRUE' }
VERSION : 0.1
   VAR_INPUT 
      IN1 : "Alarm_Parameter";
      IN2 : "Alarm_Parameter";
   END_VAR


BEGIN
	#FC_Alarm_Editiert_HMI :=
	#IN1.Hupe_Blau       <> #IN2.Hupe_Blau OR
	#IN1.Hupe_Dauer_Blau <> #IN2.Hupe_Dauer_Blau OR
	#IN1.Hupe_Dauer_Gelb <> #IN2.Hupe_Dauer_Gelb OR
	#IN1.Hupe_Dauer_Rot  <> #IN2.Hupe_Dauer_Rot OR
	#IN1.Hupe_Gelb       <> #IN2.Hupe_Gelb OR
	#IN1.La_Blau         <> #IN2.La_Blau OR
	#IN1.La_Gelb         <> #IN2.La_Gelb OR
	#IN1.La_Quit_Err <> #IN2.La_Quit_Err OR
	#IN1.nicht_Hupe_Rot  <> #IN2.nicht_Hupe_Rot OR
	#IN1.nicht_La_Rot    <> #IN2.nicht_La_Rot;
END_FUNCTION

FUNCTION "FC_OUTPUT" : Void   // FC211, STL
TITLE = Schreiben der physikalischen Ausgänge
{ S7_Optimized_Access := 'FALSE' }
AUTHOR : RE
// stored: AutoNumber false
   VAR_TEMP
      Frg_Heben_li : Bool;
      Frg_Heben_re : Bool;
      Frg_Senken_li : Bool;
      Frg_Senken_re : Bool;
      Returnwert : Int;   // Rückgabewert SFC
      RetVal : Int;
   END_VAR
BEGIN

NETWORK
TITLE = Ausgabe
// Lampen

      A     "DB_ANLAGE".BA.Simulation;
      BEC;
//Warnung
      A     "DB_Alarme".Lampe_Gelb;
      O     "DB_ANLAGE".IN.Lamp_Test;
      =     "A_Mld_Wrn";
      =     "A_Mld_Wrn(2)";
      =     "A_Mld_Wrn_Geb.G";
// Störung
      A     "DB_Alarme".Lampe_Rot;
      O     "DB_ANLAGE".IN.Lamp_Test;
      =     "A_Mld_Al";
      =     "A_Mld_Al(2)";
      =     "A_Mld_Al_Geb.G";
//Hupe
      A     "DB_ANLAGE".OUT.Stoerung_Aku;
      =     "A_Hupe";
      =     "A_Hupe(2)";
      =     "A_Hupe_Geb.G";

//Fertigmeldung 1 WT will raus: CMD = 25
      L     "DB_WT1".akt_CMD;
      L     25;
      ==I;
      A     "DB_POS".POS["DB_WT1".POS].fertig;
      O(;
      L     "DB_WT2".akt_CMD;
      ==I;
      A     "DB_POS".POS["DB_WT2".POS].fertig;
      );
      O(;
      L     "DB_WT3".akt_CMD;
      L     25;
      ==I;
      A     "DB_POS".POS["DB_WT3".POS].fertig;
      );
      O(;
      L     "DB_WT4".akt_CMD;
      ==I;
      A     "DB_POS".POS["DB_WT4".POS].fertig;
      );
      O(;
      L     "DB_WT5".akt_CMD;
      L     25;
      ==I;
      A     "DB_POS".POS["DB_WT5".POS].fertig;
      );
      O(;
      L     "DB_WT6".akt_CMD;
      ==I;
      A     "DB_POS".POS["DB_WT6".POS].fertig;
      );
      O(;
      L     "DB_WT7".akt_CMD;
      L     25;
      ==I;
      A     "DB_POS".POS["DB_WT7".POS].fertig;
      );
      O(;
      L     "DB_WT8".akt_CMD;
      ==I;
      A     "DB_POS".POS["DB_WT8".POS].fertig;
      );
      O(;
      L     "DB_WT9".akt_CMD;
      L     25;
      ==I;
      A     "DB_POS".POS["DB_WT9".POS].fertig;
      );
      O(;
      L     "DB_WT10".akt_CMD;
      ==I;
      A     "DB_POS".POS["DB_WT10".POS].fertig;
      );
      O(;
      L     "DB_WT11".akt_CMD;
      L     25;
      ==I;
      A     "DB_POS".POS["DB_WT11".POS].fertig;
      );
      O(;
      L     "DB_WT12".akt_CMD;
      ==I;
      A     "DB_POS".POS["DB_WT12".POS].fertig;
      );
      A     "Clock_1Hz";
      O     "DI_FW_Auftrag_DB".Frg_Ausfahrt;
      O     "DB_ANLAGE".IN.Lamp_Test;
      =     "A_Mld_fertig";
      =     "A_Mld_fertig(2)";
      =     "A_Mld_fertig_Geb.G";

      A     "DB_ANLAGE".OUT.Fehler_Quitt;
      O     "DB_ANLAGE".IN.Lamp_Test;
      =     "A_LED_Q_Err";
      L     3;
      JC    LED;
      L     0;
LED:  T     "MobilePanel".Drucktaster_K2_LED;

      AN    "DB_PNOZ_IN_Out".In.PNOZ_OK;
      =     "A_LED_Q_NH";

// Meldung Automatik
      A     "DB_ANLAGE".OUT.MD_Auto;
      O     "DB_ANLAGE".IN.Lamp_Test;
      =     "A_Mld_Automatik";
      =     "A_Mld_Automatik(2)";
      =     "A_Mld_Automatik_Geb.G";

// Turmleuchte Tür
      AN    "E_Wrn_Gas_ok";
      =     "A_TL_T_Vorarlarm_Gas";
      =     "A_TL_T_Vorarlarm_Gas(2)";

      AN    "E_Al_Gas_ok";
      =     "A_TL_T_Hauptalarm_Gas";
      =     "A_TL_T_Hauptalarm_Gas(2)";

      AN    "E_Al_Gas_ok";
      =     "A_TL_T_Hupe";
      =     "A_TL_T_Hupe(2)";

// Koppelsignale
// --> AWA
      SET;
      =     "A_KS_in_Betrieb";
// --> Wäscher
      AN    "E_Niv_max_CM05.BL01";
      A     "E_Niv_Uel_CM05.BL12";
      =     "A_KS_CM05_nicht_Voll";

// Werkschutz
// 14x Leckage
      A     "FP_CM02.GP04".Mld.Leckage;
      O     "Pu_CL01.GP08".Mld.Leckage;
      O     "Pu_CL02.GP09".Mld.Leckage;
      O     "Pu_GP01.GP12".Mld.Leckage;
      O     "Pu_GP02.GP07".Mld.Leckage;
      O     "Pu_GP01.GP13".Mld.Leckage_Pumpe;
      O     "Pu_GP01.GP13".Mld.Leckage_PFA_Uebergang;
      O     "Pu_GP01.GP13".Mld.Leckage_Doppelrohr;
      O     "Pu_GP01.GP13".Mld.Leckage_Uml_Tunnel;
      O     "Pu_GP02.GP10".Mld.Leckage_Pumpe;
      O     "Pu_GP02.GP10".Mld.Leckage_PFA_Uebergang;
      ON    "E_LS_GP02.BL26";
      O     "Pu_GP02.GP10".Mld.Leckage_Doppelschlauch;
      ON    "E_LS_GP02.BL33";
      =     "A_Mld_WS_Leckage";
// 3x Überlauf
      A     "UP_CM01.GP02".Mld.Niv_Ueberlauf;
      O     "UP_CM02.GP05".Mld.Niv_Ueberlauf;
      O     "Pu_CM05.GP11_DB".Mld."Uel_CM05.BL05";
      =     "A_Mld_WS_Ueberlauf";

      A     "DB_Alarme".Lampe_Rot;
      =     "A_Mld_WS_SSt";

// LED Türen
      AN    "DB_PNOZ_IN_Out".In.Tuer_VS_ok;
      A     "Clock_1Hz";
      =     "A_LED_Tuer_VS";

      AN    "DB_PNOZ_IN_Out".In.Tuer_RS_ok;
      A     "Clock_1Hz";
      =     "A_LED_Tuer_RS";


NETWORK
TITLE = FW
// Transportsystem
// Reparaturbetrieb
      A     "DB_ANLAGE".IN.Reparatur;
      A     "DB_ANLAGE".IN.BA_Tipp;
      =     "A_RepB";

//--------------------------
//FW1
//--------------------------
// FU Fahrt: FU[10]

      CALL  "FB_FU_OUT_TW", "DI_FU_Fahrt"
      ( Req_High       := "DI_FW_1".OUT.VOR,
        Req_Low        := "DI_FW_1".OUT.RUECK,
        Reglersperre   := "FU_In_Out".FU[10].PA.Steuerwort.RegSp,
        Freigabe_Stopp := "FU_In_Out".FU[10].PA.Steuerwort.FrgStop,
        Freigabe_Halt  := "FU_In_Out".FU[10].PA.Steuerwort.FrgHalt,
        Break_ok       := "DI_FW_POS_1".IN.Break_on,
        SollSpeed      := "DI_FW_POS_1".OUT.SollSpeed,
        Ist_Speed      := "DI_FW_POS_1".IN.IstSpeed,
        PAW_Speed      := "FU_In_Out".FU[10].PA.Speed,
        PEW_Speed      := "FU_In_Out".FU[10].PE.Speed
      );

      A     "DI_FW_1".OUT.VOR;
      O     "DI_FW_1".OUT.RUECK;
      =     "A_Frg_FU_Fahrt";

// FU Hub links: FU[11]
      A     "DI_FW_1".OUT.HEBEN_li;
      =     "A_Heb_li";
      A     "DI_FW_1".OUT.SENKEN_li;
      =     "A_Snk_li";

      A     "DI_FW_1".OUT.HEBEN_li;
      A     "A_RepB";
      O     "E_Frg_Heb_li";
      =     #Frg_Heben_li;

      A     "DI_FW_1".OUT.SENKEN_li;
      A     "A_RepB";
      O     "E_Frg_Snk_li";
      =     #Frg_Senken_li;

      CALL  "FB_FU_OUT_TW", "DI_FU_Hub_links"
      ( Req_High       := #Frg_Heben_li,
        Req_Low        := #Frg_Senken_li,
        Reglersperre   := "FU_In_Out".FU[11].PA.Steuerwort.RegSp,
        Freigabe_Stopp := "FU_In_Out".FU[11].PA.Steuerwort.FrgStop,
        Freigabe_Halt  := "FU_In_Out".FU[11].PA.Steuerwort.FrgHalt,
        Break_ok       := "DI_FW_HUB_links".IN.Break_on,
        SollSpeed      := "DI_FW_HUB_links".OUT.SollSpeed,
        Ist_Speed      := "DI_FW_HUB_links".IN.IstSpeed,
        PAW_Speed      := "FU_In_Out".FU[11].PA.Speed,
        PEW_Speed      := "FU_In_Out".FU[11].PE.Speed
      );

      A     "DI_FW_1".OUT.HEBEN_li;
      O     "DI_FW_1".OUT.SENKEN_li;
      =     "A_Frg_FU_Hub_li";

      A     "DI_FW_1".ZST.Tipp;
      A     "DI_FW_1".ZST.BEREIT;
      A     "DI_FW_1".ZST.Unten_li;
      A     "T_ErrQuitt";
      =     "A_WZ_Tara_li_1";
      =     "A_WZ_Tara_li_2";
      =     "A_WZ_Tara_li_3";
      =     "A_WZ_Tara_li_4";

// FU Hub rechts: FU[12]
      A     "DI_FW_1".OUT.HEBEN_re;
      =     "A_Heb_re";
      A     "DI_FW_1".OUT.SENKEN_re;
      =     "A_Snk_re";

      A     "DI_FW_1".OUT.HEBEN_re;
      A     "A_RepB";
      O     "E_Frg_Heb_re";
      =     #Frg_Heben_re;

      A     "DI_FW_1".OUT.SENKEN_re;
      A     "A_RepB";
      O     "E_Frg_Snk_re";
      =     #Frg_Senken_re;

      CALL  "FB_FU_OUT_TW", "DI_FU_Hub_rechts"
      ( Req_High       := #Frg_Heben_re,
        Req_Low        := #Frg_Senken_re,
        Reglersperre   := "FU_In_Out".FU[12].PA.Steuerwort.RegSp,
        Freigabe_Stopp := "FU_In_Out".FU[12].PA.Steuerwort.FrgStop,
        Freigabe_Halt  := "FU_In_Out".FU[12].PA.Steuerwort.FrgHalt,
        Break_ok       := "DI_FW_HUB_rechts".IN.Break_on,
        SollSpeed      := "DI_FW_HUB_rechts".OUT.SollSpeed,
        Ist_Speed      := "DI_FW_HUB_rechts".IN.IstSpeed,
        PAW_Speed      := "FU_In_Out".FU[12].PA.Speed,
        PEW_Speed      := "FU_In_Out".FU[12].PE.Speed
      );

      A     "DI_FW_1".OUT.HEBEN_re;
      O     "DI_FW_1".OUT.SENKEN_re;
      =     "A_Frg_FU_Hub_re";


      A     "DI_FW_1".ZST.Tipp;
      A     "DI_FW_1".ZST.BEREIT;
      A     "DI_FW_1".ZST.Unten_re;
      A     "T_ErrQuitt";
      =     "A_WZ_Tara_re_1";
      =     "A_WZ_Tara_re_2";
      =     "A_WZ_Tara_re_3";
      =     "A_WZ_Tara_re_4";


NETWORK
TITLE = Be- und Entladestände (QF1 / QF2)
// WR02/03
// QF 1 FU[8]

      CALL  "FB_FU_OUT_TW", "DI_FU_WR02"
      ( Req_High       := "DI_QF_WR02_03".Out.WR02_einfahren,
        Req_Low        := "DI_QF_WR02_03".Out.WR02_ausfahren,
        Reglersperre   := "FU_In_Out".FU[8].PA.Steuerwort.RegSp,
        Freigabe_Stopp := "FU_In_Out".FU[8].PA.Steuerwort.FrgStop,
        Freigabe_Halt  := "FU_In_Out".FU[8].PA.Steuerwort.FrgHalt,
        Break_ok       := ,
        SollSpeed      := "DI_QF_WR02_03".Out.Soll_speed_WR02,
        Ist_Speed      := "DI_QF_WR02_03".In.FU_speed_WR02,
        PAW_Speed      := "FU_In_Out".FU[8].PA.Speed,
        PEW_Speed      := "FU_In_Out".FU[8].PE.Speed
      );

      A     "DI_QF_WR02_03".Out.WR02_einfahren;
      O     "DI_QF_WR02_03".Out.WR02_ausfahren;
      =     "A_Frg_FU_QF_WR02";

// QF 2 FU[9]

      CALL  "FB_FU_OUT_TW", "DI_FU_WR03"
      ( Req_High       := "DI_QF_WR02_03".Out.WR03_einfahren,
        Req_Low        := "DI_QF_WR02_03".Out.WR03_ausfahren,
        Reglersperre   := "FU_In_Out".FU[9].PA.Steuerwort.RegSp,
        Freigabe_Stopp := "FU_In_Out".FU[9].PA.Steuerwort.FrgStop,
        Freigabe_Halt  := "FU_In_Out".FU[9].PA.Steuerwort.FrgHalt,
        Break_ok       := ,
        SollSpeed      := "DI_QF_WR02_03".Out.Soll_speed_WR03,
        Ist_Speed      := "DI_QF_WR02_03".In.FU_speed_WR03,
        PAW_Speed      := "FU_In_Out".FU[9].PA.Speed,
        PEW_Speed      := "FU_In_Out".FU[9].PE.Speed
      );

      A     "DI_QF_WR02_03".Out.WR03_einfahren;
      O     "DI_QF_WR02_03".Out.WR03_ausfahren;
      =     "A_Frg_FU_QF_WR03";


NETWORK
TITLE = 
// Ausgänge
      CALL  "Output_Peripherie";

END_FUNCTION

FUNCTION_BLOCK "FB_FU_OUT_TW"   // FB12, LAD
TITLE = Ausgabe Einzel-FU
{ S7_Optimized_Access := 'TRUE' }
// stored: AutoNumber false, IsIECCheckEnabled true, MemoryReserve 100, SetENOAutomatically false
   VAR_INPUT
      Req_High : Bool;   // Anforderung Vorwärts/Heben
      Req_Low : Bool;   // Anforderun Rückwärts/Senken
   END_VAR
   VAR_IN_OUT
      Reglersperre : Bool;
      Freigabe_Stopp : Bool;
      Freigabe_Halt : Bool;
      Break_ok : Bool;
      SollSpeed : Int;   // Geschwindigkeit Fahren in %
      Ist_Speed : Int;
      PAW_Speed : Int;
      PEW_Speed : Int;
   END_VAR
   VAR RETAIN
      maxSpeed : Real := 7500.0;   // maximale Ausgabe (entspricht 100%)
      Faktor { ExternalAccessible := 'False'; ExternalVisible := 'False'; ExternalWritable := 'False'} : Real := 100.0;
      minSpeed : Int := 750;   // Freigabe nehmen unterhalb diesen Wertes im PEW
   END_VAR
   VAR_TEMP
      TempSpeed : Real;
      Faktor_Sim : Real;
      Delta : Int;
   END_VAR
BEGIN

REGION Network 1 (SCL): Istwert erfassen
   REGION Istwert erfassen
       // Statement section REGION
       #Ist_Speed:=REAL_TO_INT((INT_TO_REAL(#PEW_Speed)/#maxSpeed) * #Faktor);
   END_REGION
END_REGION

REGION Network 2 (SCL): Ausgabe Speed
   REGION Ausgabe Speed

       //Not-Halt --> sofort aus
       IF "DB_ANLAGE".BA.Not_Aus THEN
           #Reglersperre := TRUE;
           #Freigabe_Stopp := FALSE;
           #PAW_Speed := 0;

           //vorwärts/hoch positive Ausgabe    
       ELSIF #Req_High AND #SollSpeed <> 0 THEN
           #Reglersperre := FALSE;
           #Freigabe_Stopp := TRUE;
           #PAW_Speed := REAL_TO_INT(INT_TO_REAL(#SollSpeed) / #Faktor * #maxSpeed);

           //rückwärts/runter negative Ausgabe    
       ELSIF #Req_Low AND #SollSpeed <> 0 THEN
           #Reglersperre := FALSE;
           #Freigabe_Stopp := TRUE;
           #PAW_Speed := REAL_TO_INT(INT_TO_REAL(#SollSpeed) / #Faktor * #maxSpeed * -1.0);

           //sonst aus    
       ELSE
           #Freigabe_Stopp := #PEW_Speed >= #minSpeed;
           #Reglersperre := FALSE;
           #PAW_Speed := 0;
       END_IF;

       #Freigabe_Halt := #Freigabe_Stopp;
       #Break_ok := NOT #Freigabe_Stopp AND #Ist_Speed=0;

   END_REGION
END_REGION

REGION Network 3 (SCL): Simulation
   REGION Simulation

       IF "DB_ANLAGE".BA.Simulation THEN

           //Abfahrrampe berechnen
           #Faktor_Sim := 15.0; //500ms von 7500 auf 0 (7500.0/500.0)
           //Korrekturwert berechnen
           #Delta := REAL_TO_INT(#Faktor_Sim * INT_TO_REAL("DI_FW_MANAGER".akt_CT));

           //Geschwindigkeit reduzieren
           IF #PEW_Speed > #PAW_Speed THEN
               #PEW_Speed := #PEW_Speed - #Delta;
               IF #PEW_Speed <= #PAW_Speed THEN
                   #PEW_Speed := #PAW_Speed;
               END_IF;

               //Geschwindigkeit erhöhen
           ELSIF #PEW_Speed < #PAW_Speed THEN
               #PEW_Speed := #PEW_Speed + #Delta;
               IF #PEW_Speed >= #PAW_Speed THEN
                   #PEW_Speed := #PAW_Speed;
               END_IF;

           ELSE
               #PEW_Speed := #PAW_Speed;
           END_IF; 

       END_IF;
   END_REGION
END_REGION
END_FUNCTION_BLOCK

FUNCTION "Output_Peripherie" : Void   // FC1011, LAD
{ S7_Optimized_Access := 'TRUE' }
// stored: AutoNumber false, SetENOAutomatically true
BEGIN

REGION Network 1 (SCL): Schnellauftor
   "A_RT_auf" := "Tor".Out.auf;
   "A_RT_zu" := "Tor".Out.zu;
END_REGION

REGION Network 2 (SCL): Deckel
   // CM01
   "A_Dkl_li_auf_CM01" := "Deckel_CM01".Out.links_auf;
   "A_Dkl_li_zu_CM01" := "Deckel_CM01".Out.links_zu;
   "A_Dkl_re_auf_CM01" := "Deckel_CM01".Out.rechts_auf;
   "A_Dkl_re_zu_CM01" := "Deckel_CM01".Out.rechts_zu;
   // CM02
   "A_Dkl_li_auf_CM02" := "Deckel_CM02".Out.links_auf;
   "A_Dkl_li_zu_CM02" := "Deckel_CM02".Out.links_zu;
   "A_Dkl_re_auf_CM02" := "Deckel_CM02".Out.rechts_auf;
   "A_Dkl_re_zu_CM02" := "Deckel_CM02".Out.rechts_zu;
END_REGION

REGION Network 3 (SCL): CM01
   //Filtern
   // Pumpe (FU[1])
   "A_Frg_FU_FP_HQ01" := "FP_CM01.GP01".Out.GP0x_Ein;

   "FU_In_Out".FU[1].PA.Steuerwort.FrgHalt := "FP_CM01.GP01".Out.GP0x_Ein;
   "FU_In_Out".FU[1].PA.Steuerwort.FrgStop := "FP_CM01.GP01".Out.GP0x_Ein;
   "FU_In_Out".FU[1].PA.Steuerwort.RegSp := NOT "FU_In_Out".FU[1].PA.Steuerwort.FrgHalt;
   "FU_In_Out".FU[1].PA.Speed := "FP_CM01.GP01".Out.Soll_speed;

   // IF ("FP_CM01.GP01".In."Betriebsart" = 0) AND ("Panel".FP_CM01.BA = 1) THEN
   //     "Panel".FP_CM01.BA := 0; // Filtern
   // END_IF;

   //Ventile
   "A_CM01.QM18" := "FP_CM01.GP01".Out.Ventil_Saugseite;
   "A_CM01.QM19" := "FP_CM01.GP01".Out.Spülventil_P_Eingang;
   "A_HQ01.LV01" := "FP_CM01.GP01".Out.Ventil_Entlueften;
   "A_HQ01.QM21" := "FP_CM01.GP01".Out.Ventil_Eingang_Filter;
   "A_HQ01.QM22" := "FP_CM01.GP01".Out.Spülventil_F_Eingang;
   "A_HQ01.QM23" := "FP_CM01.GP01".Out.Ventil_Ausgang_Filter;
   "A_HQ01.QM24" := "FP_CM01.GP01".Out.Spülventil_Ausgang;

   // Umwälzen
   // Pumpe (FU[2])
   "A_Frg_FU_UP_HF_CM01" := "UP_CM01.GP02".Out.GP0x_Ein;

   "FU_In_Out".FU[2].PA.Steuerwort.FrgHalt := "UP_CM01.GP02".Out.GP0x_Ein;
   "FU_In_Out".FU[2].PA.Steuerwort.FrgStop := "UP_CM01.GP02".Out.GP0x_Ein;
   "FU_In_Out".FU[2].PA.Steuerwort.RegSp := NOT "FU_In_Out".FU[2].PA.Steuerwort.FrgHalt;
   "FU_In_Out".FU[2].PA.Speed := "UP_CM01.GP02".Out.Soll_speed;

   //Ventile
   "A_CM01.QM25" := "UP_CM01.GP02".Out.Ventil_Saugseite;
   "A_CM01.QM26" := "UP_CM01.GP02".Out.Ventil_Druckseite;
   "A_CM01.QM20" := "UP_CM01.GP02".Out.Spülventil_Eingang;
   "A_CM01.QM27" := "UP_CM01.GP02".Out.Spülventil_Ausgang;
   "A_GP02.QM45":= "UP_CM01.GP02".Out.Entsorgung_UV02;
   "A_GP02.QM44" := "UP_CM01.GP02".Out.Ventil_UV02_GP01 OR "UP_CM02.GP05".Out.Ventil_UV02_GP01;
   "A_GP02.QM43" := "UP_CM01.GP02".Out.Ventil_UV02_GP02 OR "UP_CM02.GP05".Out.Ventil_UV02_GP02;
END_REGION

REGION Network 4 (SCL): CM02
   //Filtern
   // Pumpe (FU[4])
   "A_Frg_FU_FP_HQ02" := "FP_CM02.GP04".Out.GP0x_Ein;

   "FU_In_Out".FU[4].PA.Steuerwort.FrgHalt := "FP_CM02.GP04".Out.GP0x_Ein;
   "FU_In_Out".FU[4].PA.Steuerwort.FrgStop := "FP_CM02.GP04".Out.GP0x_Ein;
   "FU_In_Out".FU[4].PA.Steuerwort.RegSp := NOT "FU_In_Out".FU[4].PA.Steuerwort.FrgHalt;
   "FU_In_Out".FU[4].PA.Speed := "FP_CM02.GP04".Out.Soll_speed;

   // IF ("FP_CM02.GP04".In."Betriebsart" = 0) AND ("Panel".FP_CM02.BA = 1) THEN
   //     "Panel".FP_CM02.BA := 0; // Filtern
   // END_IF;

   //Ventile
   "A_CM02.QM55" := "FP_CM02.GP04".Out.Ventil_Saugseite;
   "A_CM02.QM56" := "FP_CM02.GP04".Out.Spülventil_P_Eingang;
   "A_HQ02.LV02" := "FP_CM02.GP04".Out.Ventil_Entlueften;
   "A_HQ02.QM59" := "FP_CM02.GP04".Out.Ventil_Eingang_Filter;
   "A_HQ02.QM58" := "FP_CM02.GP04".Out.Spülventil_F_Eingang;
   "A_HQ02.QM60" := "FP_CM02.GP04".Out.Ventil_Ausgang_Filter;
   "A_HQ02.QM61" := "FP_CM02.GP04".Out.Spülventil_Ausgang;

   // Umwälzen
   // Pumpe (FU[5])
   "A_Frg_FU_UP_HF_CM02" := "UP_CM02.GP05".Out.GP0x_Ein;

   "FU_In_Out".FU[5].PA.Steuerwort.FrgHalt := "UP_CM02.GP05".Out.GP0x_Ein;
   "FU_In_Out".FU[5].PA.Steuerwort.FrgStop := "UP_CM02.GP05".Out.GP0x_Ein;
   "FU_In_Out".FU[5].PA.Steuerwort.RegSp := NOT "FU_In_Out".FU[5].PA.Steuerwort.FrgHalt;
   "FU_In_Out".FU[5].PA.Speed := "UP_CM02.GP05".Out.Soll_speed;

   //Ventile
   "A_CM02.QM62" := "UP_CM02.GP05".Out.Ventil_Saugseite;
   "A_CM02.QM63" := "UP_CM02.GP05".Out.Ventil_Druckseite;
   "A_CM02.QM57" := "UP_CM02.GP05".Out.Spülventil_Eingang;
   "A_CM02.QM64" := "UP_CM02.GP05".Out.Spülventil_Ausgang;
   "A_GP02.QM46" := "UP_CM02.GP05".Out.Entsorgung_UV02;
END_REGION

REGION Network 5 (SCL): CM03
   // Pumpe (FU[3])
   "A_Frg_FU_UP_H2O_CM03" := "UP_CM03.GP03".Out.GP0x_Ein;

   "FU_In_Out".FU[3].PA.Steuerwort.FrgHalt := "UP_CM03.GP03".Out.GP0x_Ein;
   "FU_In_Out".FU[3].PA.Steuerwort.FrgStop := "UP_CM03.GP03".Out.GP0x_Ein;
   "FU_In_Out".FU[3].PA.Steuerwort.RegSp := NOT "FU_In_Out".FU[3].PA.Steuerwort.FrgHalt;
   "FU_In_Out".FU[3].PA.Speed := "UP_CM03.GP03".Out.Soll_speed;

   // Ventile
   "A_CM03.QM33" := "UP_CM03.GP03".Out.Ventil_Saugseite;
   "A_CM03.QM34" := "UP_CM03.GP03".Out.Ventil_Druckseite;
   "A_CM03.QM36" := "UP_CM03.GP03".Out.Spülventil;
   "A_CM03.QM37" := "UP_CM03.GP03".Out.Ventil_CM05;
END_REGION

REGION Network 6 (SCL): CM04
   // Pumpe (FU[6])
   "A_Frg_FU_UP_H2O_CM04" := "UP_CM04.GP06".Out.GP0x_Ein;

   "FU_In_Out".FU[6].PA.Steuerwort.FrgHalt := "UP_CM04.GP06".Out.GP0x_Ein;
   "FU_In_Out".FU[6].PA.Steuerwort.FrgStop := "UP_CM04.GP06".Out.GP0x_Ein;
   "FU_In_Out".FU[6].PA.Steuerwort.RegSp := NOT "FU_In_Out".FU[6].PA.Steuerwort.FrgHalt;
   "FU_In_Out".FU[6].PA.Speed := "UP_CM04.GP06".Out.Soll_speed;

   // Ventile
   "A_CM04.QM72" := "UP_CM04.GP06".Out.Ventil_Saugseite;
   "A_CM04.QM73" := "UP_CM04.GP06".Out.Ventil_Druckseite;
   "A_CM04.QM75" := "UP_CM04.GP06".Out.Spülventil;
   "A_CM04.QM76" := "UP_CM04.GP06".Out.Ventil_CM05;
END_REGION

REGION Network 7 (SCL): CM05
   // Pumpe
   "A_Pu_Entl_CM05" := "Pu_CM05.GP11_DB".Out.GP11_Ein;
   // Ventile
   "A_CM05.QM61" := "Pu_CM05.GP11_DB".Out.QM61;
   "A_CM05.QM62" := "Pu_CM05.GP11_DB".Out.QM62;
   "A_CM05.QM63" := "Pu_CM05.GP11_DB".Out.QM63;
   "A_CM05.QM64" := "Pu_CM05.GP11_DB".Out.QM64;
END_REGION

REGION Network 8 (SCL): CL0x
   // CL01
   // Pumpe
   "A_CL01.GP08" := "Pu_CL01.GP08".Out.GP0x_Ein;
   // Spülventil
   "A_CL01.QM51" := "Pu_CL01.GP08".Out.Spülventil;

   // CL02
   // Pumpe
   "A_CL02.GP09" := "Pu_CL02.GP09".Out.GP0x_Ein;
   // Spülventil
   "A_CL02.QM52" := "Pu_CL02.GP09".Out.Spülventil;
END_REGION

REGION Network 9 (SCL): GP01
   // Versorgung
   // Pumpe
   "A_GP01.GP13" := "Pu_GP01.GP13".Out.GP0x_Ein;
   // Ventile
   "A_GP01.QM14" := "Pu_GP01.GP13".Out.Ventil_Entsorgung;
   "A_GP01.QM15" := "Pu_GP01.GP13".Out.Ventil_Saugseite;
   "A_GP01.QM16" := "Pu_GP01.GP13".Out.Spülventil_Eingang;
   "A_GP01.QM17" := "Pu_GP01.GP13".Out.Spülventil_Ausgang;
   "A_GP01.QM18" := "Pu_GP01.GP13".Out.Ventil_Druckseite;
   "A_GP01.QM22" := "Pu_GP01.GP13".Out.Versorgung_UV01;

   "A_GP01.QM19" := "Pu_GP01.GP13".Out.UV01_CM02 OR "Pu_GP02.GP10".Out.UV01_CM02;
   "A_GP01.QM20" := "Pu_GP01.GP13".Out.UV01_CM01 OR "Pu_GP02.GP10".Out.UV01_CM01;

   // Entleeren Sumpf
   // Pumpe
   "A_GP01.GP12" := "Pu_GP01.GP12".Out.GP0x_Ein AND "DB_PNOZ_IN_Out".In.Tuer_zu_Seite_GP01 AND "DB_PNOZ_IN_Out".In.Tuer_zu_vorn_GP01;
   // Spülventil
   "A_GP01.QM23" := "Pu_GP01.GP12".Out.Spülventil AND "DB_PNOZ_IN_Out".In.Tuer_zu_Seite_GP01 AND "DB_PNOZ_IN_Out".In.Tuer_zu_vorn_GP01;
   // IBC
   "A_IBC_Vers" := "E_S_IBC_GP01.BG21";
END_REGION

REGION Network 10 (SCL): GP02
   // Versorgung
   // Pumpe
   "A_GP02.GP10" := "Pu_GP02.GP10".Out.GP0x_Ein;
   // Ventile
   "A_GP02.QM41" := "Pu_GP02.GP10".Out.Ventil_Entsorgung;
   "A_GP02.QM38" := "Pu_GP02.GP10".Out.Ventil_Saugseite;
   "A_GP02.QM39" := "Pu_GP02.GP10".Out.Spülventil_Eingang;
   "A_GP02.QM42" := "Pu_GP02.GP10".Out.Spülventil_Ausgang;
   "A_GP02.QM40" := "Pu_GP02.GP10".Out.Ventil_Druckseite;
   "A_GP01.QM21" := "Pu_GP02.GP10".Out.Versorgung_UV01;

   // Entleeren Sumpf
   // Pumpe
   "A_GP02.GP07" := "Pu_GP02.GP07".Out.GP0x_Ein AND "DB_PNOZ_IN_Out".In.Tuer_zu_vorn_GP02;
   // Spülventil
   "A_GP02.QM37" := "Pu_GP02.GP07".Out.Spülventil AND "DB_PNOZ_IN_Out".In.Tuer_zu_vorn_GP02;
   // IBC
   "A_IBC_Ents" := "E_S_IBC_GP02.BG22";
END_REGION
END_FUNCTION

FUNCTION "FU_Write" : Void
{ S7_Optimized_Access := 'TRUE' }
VERSION : 0.1
   VAR_TEMP 
      Ret_Value : Int;
      i : Int;
   END_VAR


BEGIN
	IF "DB_ANLAGE".BA.Simulation THEN
	    RETURN;
	END_IF;
	
	// Fehlerquittung
	FOR #i:= 1 TO "FU_In_Out".Anzahl DO
	    "FU_In_Out".FU[#i].PA.Steuerwort.Reset := "DB_ANLAGE".config.FP_In_Quitt AND "FU_In_Out".FU[#i].PE.Statusbyte.Stoer;
	END_FOR;
	
	// Pumpen
	#Ret_Value := DPWR_DAT(LADDR := "SEW-GW_UC01~Filterbeschickung_HQ01", RECORD := "FU_In_Out".FU[1].PA);
	#Ret_Value := DPWR_DAT(LADDR := "SEW-GW_UC01~Umwaelzung_CM01", RECORD := "FU_In_Out".FU[2].PA);
	#Ret_Value := DPWR_DAT(LADDR := "SEW-GW_UC01~Umwaelzung_CM03", RECORD := "FU_In_Out".FU[3].PA);
	#Ret_Value := DPWR_DAT(LADDR := "SEW-GW_UC01~Filterbeschickung_HQ02", RECORD := "FU_In_Out".FU[4].PA);
	#Ret_Value := DPWR_DAT(LADDR := "SEW-GW_UC01~Umwaelzung_CM02", RECORD := "FU_In_Out".FU[5].PA);
	#Ret_Value := DPWR_DAT(LADDR := "SEW-GW_UC01~Umwaelzung_CM04", RECORD := "FU_In_Out".FU[6].PA);
	// Ventilator
	#Ret_Value := DPWR_DAT(LADDR := "SEW-GW_UC01~Ventilator_Sperrluft", RECORD := "FU_In_Out".FU[7].PA);
	// QF
	#Ret_Value := DPWR_DAT(LADDR := "SEW-GW_UC06~QF_WR02", RECORD := "FU_In_Out".FU[8].PA);
	#Ret_Value := DPWR_DAT(LADDR := "SEW-GW_UC06~QF_WR03", RECORD := "FU_In_Out".FU[9].PA);
	
	// TW
	#Ret_Value := DPWR_DAT(LADDR := "SEW-GW_UC07~TW_Fahrt", RECORD := "FU_In_Out".FU[10].PA);
	#Ret_Value := DPWR_DAT(LADDR := "SEW-GW_UC07~TW_Hub_li_WR04", RECORD :="FU_In_Out".FU[11].PA);
	#Ret_Value := DPWR_DAT(LADDR := "SEW-GW_UC07~TW_Hub_re_WR05", RECORD := "FU_In_Out".FU[12].PA);
	
END_FUNCTION

FUNCTION "FC_Copy_Daten_Heraeus" : Void
{ S7_Optimized_Access := 'TRUE' }
VERSION : 0.1
   VAR_TEMP 
      i : Int;
   END_VAR


BEGIN
	REGION Leitwerte
	    "DB_Daten_Heraeus"."Leitwert_CM01.BN01" := "Panel".IW."LF_CM01.BN01";
	    "DB_Daten_Heraeus"."Leitwert_CM01.BN02" :=  "Panel".IW."LF_CM01.BN02";
	    "DB_Daten_Heraeus"."Leitwert_CM02.BN03":= "Panel".IW."LF_CM02.BN03";
	    "DB_Daten_Heraeus"."Leitwert_CM02.BN04" := "Panel".IW."LF_CM02.BN04";
	END_REGION ;
	
	REGION Druckwerte
	    "DB_Daten_Heraeus"."p_HQ01.BP01" := "Panel".IW."p_HQ01.BP01";
	    "DB_Daten_Heraeus"."p_HQ02.BP02" := "Panel".IW."p_HQ02.BP02";
	    "DB_Daten_Heraeus"."p_CM01.BP03" := "Panel".IW."p_CM01.BP03";
	    "DB_Daten_Heraeus"."p_CM01.BP04" := "Panel".IW."p_CM01.BP04";
	    "DB_Daten_Heraeus"."p_CM03.BP05" := "Panel".IW."p_CM03.BP05";
	    "DB_Daten_Heraeus"."p_CM02.BP06" := "Panel".IW."p_CM02.BP06";
	    "DB_Daten_Heraeus"."p_CM02.BP07" := "Panel".IW."p_CM02.BP07";
	    "DB_Daten_Heraeus"."p_CM04.BP08" := "Panel".IW."p_CM04.BP08";
	    "DB_Daten_Heraeus"."p_CM05.BP09" := "Panel".IW."p_CM05.BP09";
	   END_REGION
END_FUNCTION

ORGANIZATION_BLOCK "Diagnostic error interrupt"   // OB82, STL, DiagnosticErrorInterrupt
{ S7_Optimized_Access := 'FALSE' }
   VAR_TEMP
      EV_CLASS : Byte;   // 16#39: Event class 3, Entering event state, Internal fault event
      FLT_ID : Byte;   // Fault identifier
      PRIORITY : Byte;   // Priority of OB Execution
      OB_NUMBR : Byte;   // OB number
      RESERVED_1 : Byte;   // Reserved for system
      IO_FLAG : Byte;   // 16#54:input, 16#55:output, 16#0:not available
      MDL_ADDR : Word;   // Hardware identifier
      MDL_DEFECT : Bool;   // Module defective
      INT_FAULT : Bool;   // Internal fault
      EXT_FAULT : Bool;   // External fault
      PNT_INFO : Bool;   // Channel fault
      EXT_VOLTAGE : Bool;   // External voltage low
      FLD_CONNCTR : Bool;   // Field wiring connector missing
      NO_CONFIG : Bool;   // Module has no configuration data
      CONFIG_ERR : Bool;   // Module has configuration error
      MDL_TYPE : Byte;   // Type of module
      SUB_MDL_ERR : Bool;   // Sub-Module is missing or has error
      COMM_FAULT : Bool;   // Communication fault
      MDL_STOP : Bool;   // Module is stopped
      WTCH_DOG_FLT : Bool;   // Watch dog timer stopped module
      INT_PS_FLT : Bool;   // Internal power supply fault
      PRIM_BATT_FLT : Bool;   // Primary battery is in fault
      BCKUP_BATT_FLT : Bool;   // Backup battery is in fault
      RESERVED_2 : Bool;   // Reserved for system
      RACK_FLT : Bool;   // Rack fault, only for bus interface module
      PROC_FLT : Bool;   // Processor fault
      EPROM_FLT : Bool;   // EPROM fault
      RAM_FLT : Bool;   // RAM fault
      ADU_FLT : Bool;   // ADU fault
      FUSE_FLT : Bool;   // Fuse fault
      HW_INTR_FLT : Bool;   // Hardware interrupt input in fault
      RESERVED_3 : Bool;   // Reserved for system
      DATE_TIME : Date_And_Time;   // Date and time OB82 started
   END_VAR
BEGIN
END_ORGANIZATION_BLOCK

ORGANIZATION_BLOCK "IO access error"   // OB122, STL, IOAccessError
{ S7_Optimized_Access := 'FALSE' }
   VAR_TEMP
      EV_CLASS : Byte;   // 16#29: Event class 2, Entering event state, Internal fault event
      SW_FLT : Byte;   // 16#42:reading, 16#43:writing
      PRIORITY : Byte;   // Priority of OB Execution
      OB_NUMBR : Byte;   // OB number
      BLK_TYPE : Byte;   // 16#88:OB, 16#8C:FC, 16#8E:FB: Type of block causing the error
      MEM_AREA : Byte;   // Memory area and access type
      MEM_ADDR : Word;   // Memory address where access error occured
      BLK_NUM : Word;   // Block number in which error occured
      PRG_ADDR : Word;   // Program address where error occured
      DATE_TIME : Date_And_Time;   // Date and time OB started
   END_VAR
BEGIN
END_ORGANIZATION_BLOCK

ORGANIZATION_BLOCK "Pull or plug of modules"   // OB83, STL, PullOrPlugOfModules
{ S7_Optimized_Access := 'FALSE' }
   VAR_TEMP
      EV_CLASS : Byte;   // 16#38:Event class 3 - module inserted, 16#39: Event class 3 - module removed
      FLT_ID : Byte;   // Fault identifier
      PRIORITY : Byte;   // Priority of OB Execution
      OB_NUMBR : Byte;   // OB number
      RESERVED_1 : Byte;   // Reserved for system
      MDL_ID : Byte;   // 16#54:input, 16#55:output, 16#0:not available
      MDL_ADDR : Word;   // Hardware identifier
      RACK_NUM : Int;   // Rack number
      MDL_TYPE : Word;   // Module type
      DATE_TIME : Date_And_Time;   // Date and time OB started
   END_VAR
BEGIN
END_ORGANIZATION_BLOCK

ORGANIZATION_BLOCK "Rack or station failure"   // OB86, STL, RackOrStationFailure
TITLE = "Loss Of Rack Fault"
{ S7_Optimized_Access := 'FALSE' }
AUTHOR : RE
VERSION : 0.0
   VAR_TEMP
      OB86_EV_CLASS : Byte;   // 16#38/39 Event class 3
      OB86_FLT_ID : Byte;   // 16#C1/C4/C5, Fault identification code
      OB86_PRIORITY : Byte;   // 26/28 (Priority of 1 is lowest)
      OB86_OB_NUMBR : Byte;   // 86 (Organization block 86, OB86)
      OB86_RESERVED_1 : Byte;   // Reserved for system
      OB86_RESERVED_2 : Byte;   // Reserved for system
      OB86_MDL_ADDR : Word;   // Depending on fault identification code
      OB86_Z23 : DWord;   // see Context Help OB86
      OB86_DATE_TIME : Date_And_Time;   // Date and time OB86 started
      E_Param : DWord;
      RetVal : Int;
      DP_Slave_Nr : Int;
      Status : Array[0..1023] of Bool;
      Count : Int;
      Station_OK : Bool;
   END_VAR
BEGIN

NETWORK
TITLE = Wird bei DP-Stationsausfall und Rackfehler aktiviert
      AN    "DB_ANLAGE".IN.Watch_Profibus;  //keine Überwachung Profibus!
      BEC;

//DP-Slave Nummer
      L     #OB86_Z23.%W0;  //Nr. der DP Station (Bit 0-7 in OB86_Z23)
      AW    w#16#3ff;
      T     #DP_Slave_Nr;

//Fehler kommt/geht
      L     #OB86_EV_CLASS;
      L     16#39;  //kommendes Ereignis
      ==I;
      JC    kommt;

      L     #OB86_EV_CLASS;
      L     16#38;  //gehendes Ereignis
      ==I;
      JC    geht;

      BE;

NETWORK
TITLE = Fehler kommt
kommt:L     #OB86_FLT_ID;
      L     16#Cb;  //Ausfall einer DP-Station Code C4 Profinet CB
      <>I;
      BEC;

      L     #DP_Slave_Nr;
      SLD   3;
      LAR1;
      OPN   "DB_DP_Error";
      L     3;
      T     DBB [AR1, P#0.0];

      BE;

NETWORK
TITLE = Fehler geht
geht: L     #OB86_FLT_ID;
      L     16#Cb;  //Ausfall einer DP-Station gehendes Ereignis
      <>I;
      BEC;
      =     #Station_OK;

      L     #DP_Slave_Nr;
      SLD   3;
      LAR1;
      OPN   "DB_DP_Error";

      L     1;
      T     DBB [AR1, P#0.0];

// Check ob gestört
      CALL  DeviceStates
      ( LADDR   := "Local~PROFINET_IO-System",
        MODE    := 2,  // 2: IO-Devices/DP-Slaves gestört
        Ret_Val := #RetVal,
        STATE   := #Status
      );

//------------------------------------------------------------------------------
//Ergebnis abspeichern
      L     0;
      T     #Count;

      L     P##Status;
      LAR1;
      L     0;
retS: +AR1;

      AN    L [AR1, P#0.0];  //Laufendes Bit für Bus-Adresse
      JC    notS;

      L     #Count;
      T     "DB_DP_Error".HiAdr;  //höchste Adresse speichern
      SLD   3;
      LAR2;
      OPN   "DB_DP_Error";
      L     DBB [AR2, P#0.0];
      L     1;
      <>I;
      JC    notS;
      L     2;  //Station gestört
      T     DBB [AR2, P#0.0];

notS: L     #Count;
      +     1;
      T     #Count;
      L     1023;
      <D;
      L     P#0.1;
      JC    retS;
//------------------------------------------------------------------------------

      BE;
END_ORGANIZATION_BLOCK

ORGANIZATION_BLOCK "Startup"   // OB100, STL, Startup
TITLE = "Complete Restart"
{ S7_Optimized_Access := 'FALSE' }
AUTHOR : MS
VERSION : 0.0
// stored: AutoNumber false
   VAR_TEMP
      OB100_EV_CLASS : Byte;   // 16#13, Event class 1, Entering event state, Event logged in diagnostic buffer
      OB100_STRTUP : Byte;   // 16#81/82/83/84 Method of startup
      OB100_PRIORITY : Byte;   // 27 (Priority of 1 is lowest)
      OB100_OB_NUMBR : Byte;   // 100 (Organization block 100, OB100)
      OB100_RESERVED_1 : Byte;   // Reserved for system
      OB100_RESERVED_2 : Byte;   // Reserved for system
      OB100_STOP : Word;   // Event that caused CPU to stop (16#4xxx)
      OB100_STRT_INFO : DWord;   // Information on how system started
      OB100_DATE_TIME : Date_And_Time;   // Date and time OB100 started
      DB_Nr : DB_ANY;
      RetVal : Int;
      DB_leng : UDInt;
      Writ_Prot : Bool;
      DelVal : Int;
      attrib : Byte;
      REQ : Bool;
      Count : Int;
      aDateTime : Date_And_Time;   // aktuelle Uhrzeit
      Status : Array[0..1023] of Bool;
   END_VAR
BEGIN

NETWORK
TITLE = Not-Aus ist betätigt
//---------------------------
//Neustart-Information setzen
//---------------------------
      SET;
      R     "DB_ANLAGE".BA.Not_Aus;
      R     "DB_ANLAGE".BA.Tippbetrieb;
      R     "DB_ANLAGE".BA.Handbetrieb;
      S     "DB_ANLAGE".BA.Automat_aus;
      R     "DB_ANLAGE".BA.Automat_ein;
      S     "DB_ANLAGE".BA.FP_Automat_ein;
      S     "DB_ANLAGE".BA.COM_RST;

//---------------------------
//Initialisierung der Anlage
//---------------------------
noTime:NOP   0;

      CALL  "FC_newConfig"
      ( Anlauf := TRUE
      );

      L     S5T#5S;
      CLR;
      Pulse "T_Anlauf";
      SET;
      Pulse "T_Anlauf";
wait: NOP   0;
      A     "T_Anlauf";
      JC    wait;



NETWORK
TITLE = Verbindungsaufbau PNOZ initieren
      L     0;  // --> OFF
      T     "DB_PNOZ_Comm".Global_Status;
      SET;
      R     "DB_PNOZ_Comm".connection.activate;
      R     "DB_PNOZ_Comm".connection.established;

NETWORK
TITLE = DP-Slave-Diagnose
//==============================================================================
//Test ist Prüfung gefordert/möglich?
//Soll der Profibus überprüft werden? Dann OB86,OB100,FC203,DB203 prüfen!
      AN    "DB_ANLAGE".config.Check_Profibus;
      JC    endP;

//Prüfen ob Diagnose möglich! Ist Diagnosebaustein vorhanden?
      L     203;  //"DB_DP_Error"
      T     #DB_Nr;

      CALL  ATTR_DB
      ( REQ       := 1,
        DB_NUMBER := #DB_Nr,
        RET_VAL   := #RetVal,
        DB_LENGTH := #DB_leng,
        ATTRIB    := #attrib
      );

      L     #DB_leng;  //Baustein ist lang genug
      L     2052;  //zweimal 1024 Byte + 4 Arbeitsbytes
      <I;
      O(;
      L     #RetVal;  //Es ist ein Fehler aufgetreten
      L     0;
      <>I;
      );
      R     "DB_ANLAGE".IN.Watch_Profibus;
      JC    endP;
      S     "DB_ANLAGE".IN.Watch_Profibus;  //Überwachung möglich!!
//==============================================================================

//==============================================================================
//DB initialisieren
      L     0;
      T     #DelVal;

      CALL  FILL
      ( BVAL    := #DelVal,
        RET_VAL := #RetVal,
        BLK     := "DB_DP_Error".DP_Slave
      );

      CALL  FILL
      ( BVAL    := #DelVal,
        RET_VAL := #RetVal,
        BLK     := "DB_DP_Error".Altwert
      );

      SET;
      S     "DB_DP_Error".Init;
      R     "DB_DP_Error".Sammelstoerung;
      R     "DB_DP_Error".Sammelwarnung;
//==============================================================================

//==============================================================================
//Istausbau DP Slaves Mastersystem 1 auslesen
//------------------------------------------------------------------------------
//Lesevorgang
r_is: NOP   0;
      CALL  DeviceStates
      ( LADDR   := "Local~PROFINET_IO-System",
        MODE    := 4,  // 4: IO-Devices/DP-Slaves vorhanden
        Ret_Val := #RetVal,
        STATE   := #Status  //ein Bit je Geräte-Nr (HWconfig)
      );
//------------------------------------------------------------------------------
//------------------------------------------------------------------------------
//Ergebnis abspeichern
      L     0;
      T     #Count;

      L     P##Status;
      LAR1;
      L     0;
retI: +AR1;

      AN    L [AR1, P#0.0];  //Laufendes Bit für Bus-Adresse
      JC    notI;

      L     #Count;
      T     "DB_DP_Error".HiAdr;  //höchste Adresse speichern
      SLD   3;
      LAR2;
      OPN   "DB_DP_Error";
      L     1;
      T     DBB [AR2, P#0.0];

notI: L     #Count;
      +     1;
      T     #Count;
      L     1023;
      <D;
      L     P#0.1;
      JC    retI;
//------------------------------------------------------------------------------
//==============================================================================

//==============================================================================
//Sollausbau / Projektierung DP Slaves Mastersystem 1
//------------------------------------------------------------------------------
//Lesevorgeng
r_so: NOP   0;

      CALL  DeviceStates
      ( LADDR   := "Local~PROFINET_IO-System",
        MODE    := 1,  //1: IO-Devices/DP-Slaves sind konfiguriert
        Ret_Val := #RetVal,
        STATE   := #Status
      );

//------------------------------------------------------------------------------

//------------------------------------------------------------------------------
//projektierte Teilnehmer aufnehmen
      L     0;
      T     #Count;

      L     P##Status;
      LAR1;
      L     0;
retS: +AR1;

      AN    L [AR1, P#0.0];  //Laufendes Bit für Bus-Adresse
      JC    notS;

      L     #Count;
      L     "DB_DP_Error".HiAdr;  //höchste Adresse evtl. korrigieren
      <=I;
      JC    nKor;
      L     #Count;
      T     "DB_DP_Error".HiAdr;  //höchste Adresse evtl. korrigieren

nKor: L     #Count;
      SLD   3;
      LAR2;
      OPN   "DB_DP_Error";
      L     DBB [AR2, P#0.0];
      L     1;
      ==I;
      JC    notS;
      L     3;
      T     DBB [AR2, P#0.0];

notS: L     #Count;
      +     1;
      T     #Count;
      L     1023;
      <D;
      L     P#0.1;
      JC    retS;
//------------------------------------------------------------------------------
//==============================================================================

endP: NOP   0;

END_ORGANIZATION_BLOCK

ORGANIZATION_BLOCK "Time error interrupt"   // OB80, STL, TimeErrorInterrupt
{ S7_Optimized_Access := 'FALSE' }
   VAR_TEMP
      EV_CLASS : Byte;   // 16#35: Event class 3, Entering event state, Internal fault event
      FLT_ID : Byte;   // Fault identifier
      PRIORITY : Byte;   // Priority of OB Execution
      OB_NUMBR : Byte;   // OB number
      RESERVED_1 : Byte;   // Reserved for system
      RESERVED_2 : Byte;   // Reserved for system
      ERROR_INFO : Word;   // Error information on event
      ERR_EV_CLASS : Byte;   // Class of event causing the error
      ERR_EV_NUM : Byte;   // Number of event causing the error
      OB_PRIORITY : Byte;   // Priority of OB causing the error
      OB_NUM : Byte;   // Number of OB causing the error
      DATE_TIME : Date_And_Time;   // Date and time OB started
   END_VAR
BEGIN
END_ORGANIZATION_BLOCK

FUNCTION "Ergebnis_DT" : Void   // FC340, LAD
TITLE = Ergebnis speichern
{ S7_Optimized_Access := 'TRUE' }
// stored: AutoNumber false, SetENOAutomatically false
   VAR_INPUT
      "Name" : String;
      akt_Zeit : DTL;
      ok : Bool;
      Fehler : Bool;
   END_VAR
   VAR_TEMP
      i : Int;
   END_VAR
BEGIN

REGION Network 1 (SCL)
   //Index erhöhen
   "Drucktest".akt_Index := "Drucktest".akt_Index + 1;
   IF "Drucktest".akt_Index > 100 THEN
       "Drucktest".akt_Index := 1;
   END_IF;
   #i := "Drucktest".akt_Index;
   // --> Speichern
   "Drucktest".Ergebnis[#i].Name := #Name;

   "Drucktest".Ergebnis[#i].Zeit := #akt_Zeit;

   "Drucktest".Ergebnis[#i].ok := #ok;

   "Drucktest".Ergebnis[#i].Fehler := #Fehler;
END_REGION
END_FUNCTION

FUNCTION "FC_Anf_BE" : Void   // FC31, LAD
TITLE = Anforderung WR02 /WR03 in Automatik
{ S7_Optimized_Access := 'TRUE' }
// stored: AutoNumber false, SetENOAutomatically false
   VAR_INPUT
      Req_GO_Ausfahrt : Bool;
      Req_GO_Aufgabe : Bool;
   END_VAR
   VAR_IN_OUT
      Req_WR02_IN : Bool;
      Req_WR02_OUT : Bool;
      Req_WR03_IN : Bool;
      Req_WR03_OUT : Bool;
   END_VAR
   VAR_TEMP
      alles_frei : Bool;
      Korb_in_Anlage : Bool;
      BE1_inA : Bool;
      BE1_outA : Bool;
      BE2_inA : Bool;
      BE2_outA : Bool;
      BE3_inA : Bool;
      BE3_outA : Bool;
      BE4_inA : Bool;
      BE4_outA : Bool;
      BE5_inA : Bool;
      BE5_outA : Bool;
      BE6_inA : Bool;
      BE6_outA : Bool;
      links_ok : Bool;
      rechts_ok : Bool;
      WT_DB_Nr : Word;
   END_VAR
BEGIN

REGION Network 1 (SCL): Check Zustand
   // Hat was zu tun
   IF (#Req_WR02_IN OR #Req_WR02_OUT) OR (#Req_WR03_IN OR #Req_WR03_OUT) THEN
       RETURN;
   END_IF;
   // TW hat Befehl
   IF "DB_POS".POS[25].Quelle OR "DB_POS".POS[25].Ziel OR "DB_POS".POS[26].Quelle OR "DB_POS".POS[26].Ziel OR
       "DB_POS".POS[27].Quelle OR "DB_POS".POS[27].Ziel OR "DB_POS".POS[28].Quelle OR "DB_POS".POS[28].Ziel OR
       "DB_POS".POS[29].Quelle OR "DB_POS".POS[29].Ziel OR "DB_POS".POS[30].Quelle OR "DB_POS".POS[30].Ziel THEN
       RETURN;
   END_IF;

   // Kompleett leer
   #alles_frei := NOT "DB_BE_Stand".Stand[1].IN_Belegt AND NOT "DB_BE_Stand".Stand[2].IN_Belegt AND
   NOT "DB_BE_Stand".Stand[3].IN_Belegt AND NOT "DB_BE_Stand".Stand[4].IN_Belegt AND
   NOT "DB_BE_Stand".Stand[5].IN_Belegt AND NOT "DB_BE_Stand".Stand[6].IN_Belegt;
   // mindestens 1 Korb in der Anlage
   #Korb_in_Anlage := ("DB_POS".POS[1].next_WT + "DB_POS".POS[2].next_WT + "DB_POS".POS[3].next_WT + "DB_POS".POS[4].next_WT + "DB_POS".POS[5].next_WT + "DB_POS".POS[6].next_WT
       + "DB_POS".POS[7].next_WT + "DB_POS".POS[8].next_WT + "DB_POS".POS[9].next_WT + "DB_POS".POS[10].next_WT + "DB_POS".POS[11].next_WT + "DB_POS".POS[12].next_WT
       + "DB_POS".POS[13].next_WT + "DB_POS".POS[14].next_WT + "DB_POS".POS[15].next_WT + "DB_POS".POS[16].next_WT +"DB_POS".POS[17].next_WT + "DB_POS".POS[18].next_WT
       + "DB_POS".POS[19].next_WT + "DB_POS".POS[20].next_WT + "DB_POS".POS[21].next_WT + "DB_POS".POS[22].next_WT +"DB_POS".POS[23].next_WT + "DB_POS".POS[24].next_WT
       ) > 0;
END_REGION

NETWORK
TITLE = in die Anlage / aus der Anlage ?
      L     0;
      L     "DB_POS".POS[25].WT_DB;
      >=I;
      R     #BE1_inA;
      R     #BE1_outA;
      JC    BE_2;
      L     "DB_POS".POS[25].WT_DB;
      +     +100;
      T     #WT_DB_Nr;
      OPN   DB [#WT_DB_Nr];
      A     %DBX18.1;  //"DB_WTx".in_Anlage
      S     #BE1_inA;
      R     #BE1_outA;
      JC    BE_2;
      A     %DBX18.3;  //"DB_WTx".aus_Anlage
      S     #BE1_outA;
      R     #BE1_inA;

BE_2: L     0;
      L     "DB_POS".POS[26].WT_DB;
      >=I;
      R     #BE2_inA;
      R     #BE2_outA;
      JC    BE_3;
      L     "DB_POS".POS[26].WT_DB;
      +     +100;
      T     #WT_DB_Nr;
      OPN   DB [#WT_DB_Nr];
      A     %DBX18.1;  //"DB_WTx".in_Anlage
      S     #BE2_inA;
      R     #BE2_outA;
      JC    BE_3;
      A     %DBX18.3;  //"DB_WTx".aus_Anlage
      S     #BE2_outA;
      R     #BE2_inA;

BE_3: L     0;
      L     "DB_POS".POS[27].WT_DB;
      >=I;
      R     #BE3_inA;
      R     #BE3_outA;
      JC    BE_4;
      L     "DB_POS".POS[27].WT_DB;
      +     +100;
      T     #WT_DB_Nr;
      OPN   DB [#WT_DB_Nr];
      A     %DBX18.1;  //"DB_WTx".in_Anlage
      S     #BE3_inA;
      R     #BE3_outA;
      JC    BE_4;
      A     %DBX18.3;  //"DB_WTx".aus_Anlage
      S     #BE3_outA;
      R     #BE3_inA;

BE_4: L     0;
      L     "DB_POS".POS[28].WT_DB;
      >=I;
      R     #BE4_inA;
      R     #BE4_outA;
      JC    BE_5;
      L     "DB_POS".POS[28].WT_DB;
      +     +100;
      T     #WT_DB_Nr;
      OPN   DB [#WT_DB_Nr];
      A     %DBX18.1;  //"DB_WTx".in_Anlage
      S     #BE4_inA;
      R     #BE4_outA;
      JC    BE_5;
      A     %DBX18.3;  //"DB_WTx".aus_Anlage
      S     #BE4_outA;
      R     #BE4_inA;

BE_5: L     0;
      L     "DB_POS".POS[29].WT_DB;
      >=I;
      R     #BE5_inA;
      R     #BE5_outA;
      JC    BE_6;
      L     "DB_POS".POS[29].WT_DB;
      +     +100;
      T     #WT_DB_Nr;
      OPN   DB [#WT_DB_Nr];
      A     %DBX18.1;  //"DB_WTx".in_Anlage
      S     #BE5_inA;
      R     #BE5_outA;
      JC    BE_6;
      A     %DBX18.3;  //"DB_WTx".aus_Anlage
      S     #BE5_outA;
      R     #BE5_inA;

BE_6: L     0;
      L     "DB_POS".POS[30].WT_DB;
      >=I;
      R     #BE6_inA;
      R     #BE6_outA;
      JC    BE_E;
      L     "DB_POS".POS[30].WT_DB;
      +     +100;
      T     #WT_DB_Nr;
      OPN   DB [#WT_DB_Nr];
      A     %DBX18.1;  //"DB_WTx".in_Anlage
      S     #BE6_inA;
      R     #BE6_outA;
      JC    BE_E;
      A     %DBX18.3;  //"DB_WTx".aus_Anlage
      S     #BE6_outA;
      R     #BE6_inA;

BE_E: NOP   0;


REGION Network 3 (SCL): Großoptik
   IF #Req_GO_Ausfahrt  OR #BE3_outA  OR #BE4_outA THEN
       // Warten auf Korb
       IF "DB_BE_Stand".Stand[3].IN_innen AND #alles_frei THEN
           RETURN;
       END_IF;
       // Fertigware Raus
       #links_ok := #BE3_outA AND NOT #BE4_inA AND NOT #BE2_inA AND NOT #BE6_inA;

       #rechts_ok := #BE4_outA AND NOT #BE3_inA AND NOT #BE1_inA AND NOT #BE5_inA;

       IF "DB_BE_Stand".Stand[3].IN_innen AND (#links_ok OR #rechts_ok) THEN
           #Req_WR02_OUT := #Req_WR03_OUT :=TRUE;
           RETURN;
       END_IF;
       // Leer Rein
       IF NOT "DB_BE_Stand".Stand[3].IN_innen AND #alles_frei THEN
           #Req_WR02_IN := #Req_WR03_IN := TRUE;
           RETURN;
       END_IF;
    END_IF;

    IF #Req_GO_Aufgabe OR #BE3_inA  OR #BE4_inA  THEN
        // Warten auf Korb
        IF "DB_BE_Stand".Stand[3].IN_aussen AND #alles_frei THEN
            RETURN;
        END_IF;
        // Rohware --> Rein BE3 / BE4
        #links_ok := #BE3_inA AND "DB_BE_Stand".Stand[3].IN_Freigabe AND NOT #BE4_outA
        AND (#BE2_inA AND  "DB_BE_Stand".Stand[2].IN_Freigabe OR NOT "DB_BE_Stand".Stand[2].IN_Belegt)
        AND (#BE6_inA AND  "DB_BE_Stand".Stand[6].IN_Freigabe OR NOT "DB_BE_Stand".Stand[6].IN_Belegt);

        #rechts_ok := #BE4_inA AND "DB_BE_Stand".Stand[4].IN_Freigabe AND NOT #BE3_outA
        AND (#BE1_inA AND  "DB_BE_Stand".Stand[1].IN_Freigabe OR NOT "DB_BE_Stand".Stand[1].IN_Belegt)
        AND (#BE5_inA AND  "DB_BE_Stand".Stand[5].IN_Freigabe OR NOT "DB_BE_Stand".Stand[5].IN_Belegt);

        IF "DB_BE_Stand".Stand[3].IN_aussen AND (#links_ok OR #rechts_ok) THEN
            #Req_WR02_IN := #Req_WR03_IN := TRUE;
            RETURN;
        END_IF;
        // Leer Raus
        IF NOT "DB_BE_Stand".Stand[3].IN_aussen AND #alles_frei THEN
            #Req_WR02_OUT := #Req_WR03_OUT := TRUE;
            RETURN;
        END_IF;
    END_IF;
END_REGION

REGION Network 4 (SCL): Schmalware (kurz oder lang)
   // Warten auf Korb
   IF #alles_frei AND (("DB_BE_Stand".Stand[1].IN_aussen AND "DB_BE_Stand".Stand[5].IN_innen) OR ("DB_BE_Stand".Stand[5].IN_aussen AND "DB_BE_Stand".Stand[1].IN_innen)) THEN
       RETURN;
   END_IF;

   // Fertigware Raus BE1
   IF "DB_BE_Stand".Stand[1].IN_innen AND ((#BE1_outA AND NOT #BE2_inA) OR (#BE2_outA AND NOT #BE1_inA)) THEN
       #Req_WR02_OUT := TRUE;
       IF "DB_BE_Stand".Stand[5].IN_aussen AND NOT "DB_BE_Stand".Stand[5].IN_Belegt AND NOT "DB_BE_Stand".Stand[6].IN_Belegt AND #Korb_in_Anlage THEN
           #Req_WR03_IN := TRUE;
       END_IF;
       RETURN;
   END_IF;
   // Fertigware Raus BE5
   IF "DB_BE_Stand".Stand[5].IN_innen AND ((#BE5_outA AND NOT #BE6_inA) OR (#BE6_outA AND NOT #BE5_inA)) THEN
       #Req_WR03_OUT := TRUE;
       IF "DB_BE_Stand".Stand[1].IN_aussen AND NOT "DB_BE_Stand".Stand[1].IN_Belegt AND NOT "DB_BE_Stand".Stand[2].IN_Belegt AND #Korb_in_Anlage THEN
           #Req_WR02_IN := TRUE;
       END_IF;
       RETURN;
   END_IF;
   // Rohware --> Rein BE1 / BE2
   IF "DB_BE_Stand".Stand[1].IN_aussen AND ((#BE1_inA AND "DB_BE_Stand".Stand[1].IN_Freigabe AND NOT #BE2_outA) OR (#BE2_inA AND "DB_BE_Stand".Stand[2].IN_Freigabe AND NOT #BE1_outA)) THEN
       #Req_WR02_IN := TRUE;
       IF "DB_BE_Stand".Stand[5].IN_innen AND NOT "DB_BE_Stand".Stand[5].IN_Belegt AND NOT "DB_BE_Stand".Stand[6].IN_Belegt THEN
           #Req_WR03_OUT := TRUE;
       END_IF;
       RETURN;
   END_IF;
   // Rohware --> Rein BE5 / BE6
   IF "DB_BE_Stand".Stand[5].IN_aussen AND ((#BE5_inA AND "DB_BE_Stand".Stand[5].IN_Freigabe AND NOT #BE6_outA) OR (#BE6_inA AND "DB_BE_Stand".Stand[6].IN_Freigabe AND  NOT #BE5_outA)) THEN
       #Req_WR03_IN := TRUE;
       IF "DB_BE_Stand".Stand[1].IN_innen AND NOT "DB_BE_Stand".Stand[1].IN_Belegt AND NOT "DB_BE_Stand".Stand[2].IN_Belegt THEN
           #Req_WR02_OUT := TRUE;
       END_IF;
       RETURN;
   END_IF;

   // Beide drin 
   IF "DB_BE_Stand".Stand[1].IN_innen AND "DB_BE_Stand".Stand[5].IN_innen THEN
       IF NOT "DB_BE_Stand".Stand[1].IN_Belegt AND NOT "DB_BE_Stand".Stand[2].IN_Belegt AND NOT "DB_BE_Stand".Stand[3].IN_Belegt AND NOT "DB_BE_Stand".Stand[4].IN_Belegt THEN
           #Req_WR02_OUT := TRUE;
           RETURN;
       END_IF;
       IF NOT "DB_BE_Stand".Stand[5].IN_Belegt AND NOT "DB_BE_Stand".Stand[6].IN_Belegt AND NOT "DB_BE_Stand".Stand[3].IN_Belegt AND NOT "DB_BE_Stand".Stand[4].IN_Belegt THEN
           #Req_WR03_OUT := TRUE;
           RETURN;
       END_IF;
   END_IF;

   // Beide draussen und min. 1 Korb in Anlage
   IF "E_T_Frg_BE" AND "DB_BE_Stand".Stand[1].IN_aussen AND "DB_BE_Stand".Stand[5].IN_aussen AND #Korb_in_Anlage THEN
       IF NOT "DB_BE_Stand".Stand[1].IN_Belegt AND NOT "DB_BE_Stand".Stand[2].IN_Belegt AND NOT "DB_BE_Stand".Stand[3].IN_Belegt AND NOT "DB_BE_Stand".Stand[4].IN_Belegt THEN
           #Req_WR02_IN := TRUE;
           RETURN;
       END_IF;
       IF NOT "DB_BE_Stand".Stand[5].IN_Belegt AND NOT "DB_BE_Stand".Stand[6].IN_Belegt AND NOT "DB_BE_Stand".Stand[3].IN_Belegt AND NOT "DB_BE_Stand".Stand[4].IN_Belegt THEN
           #Req_WR03_IN := TRUE;
           RETURN;
       END_IF;
   END_IF;
END_REGION
END_FUNCTION

FUNCTION "FC_EXPO_TIME" : Void   // FC5, STL
TITLE = EXPOSITIONSZEIT
{ S7_Optimized_Access := 'FALSE' }
AUTHOR : MS
// Taktet die Expositionszeit aller aktiven Positionen herunter.
// stored: AutoNumber false, ParameterPassing true
   VAR_TEMP
      anzahl : Int;
      maxPos : Int;
      ok : Bool;
      Count : Int;
      X_DB : Word;
      poin : DWord;
      Taktzeit_typ : Int;
      Taktzeit_akt : Int;
      Systemzeit : DInt;
      WT_DB : Int;
   END_VAR
BEGIN

NETWORK
TITLE = TAKT
// Im Takt wird die Expozeit um 1 herunter gezählt.
// Die Zeit, welche dieser Wert bedeutet ist im OB35 einstellbar.
// Ein Vielfaches von 100ms (Weckalarmzeit) ist dort notwendig.

      L     "DB_ANLAGE".config.ANZ_FW;
retF: T     #Count;
      L     0;
      <=I;
      JC    QT;

      L     #Count;
      L     10;
      +I;
      T     #X_DB;

      OPN   DB [#X_DB];
      L     0;
      L     %DBD46;  //"DBI_FW_1".ZST.Rest_Zeit
      >=D;
      O     %DBX0.2;  //"DBI_FW_1".ZST.FEHLER
      JC    FX;
      +     DINT#-1;
      T     %DBD46;  //"DBI_FW_1".ZST.Rest_Zeit

FX:   AN    %DBX394.6;  //"DI_FW_1".TMP.FW_gestartet
      O     %DBX0.2;  //"DI_FW_1".ZST.FEHLER
      JC    nexF;
      L     %DBD34;  //"DI_FW_1".ZST.Verweil
      +     1;
      T     %DBD34;  //"DI_FW_1".ZST.Verweil

      AN    %DBX68.0;  //"DI_FW_1".OUT.VOR
      AN    %DBX68.1;  //"DI_FW_1".OUT.RUECK
      AN    %DBX68.3;  //"DI_FW_1".OUT.HEBEN
      AN    %DBX68.4;  //"DI_FW_1".OUT.SENKEN
      JC    nexF;
      L     %DBD382;  //"DI_FW_1".TMP.Dauer
      +     DINT#1;
      T     %DBD382;  //"DI_FW_1".TMP.Dauer

nexF: L     #Count;
      L     1;
      -I;
      JC    retF;


QT:   L     "DB_ANLAGE".config.ANZ_QT;
retQ: T     #Count;
      L     0;
      <=I;
      JC    wtr;

      L     #Count;
      L     30;
      +I;
      T     #X_DB;

      OPN   DB [#X_DB];

      L     0;
      L     %DBD46;  //"DBI_QT_1".IN.Count_LokHand
      >=D;
      JC    QTx;
      L     1;
      -D;
      T     %DBD46;  //"DBI_QT_1".IN.Count_LokHand
QTx:  A     %DBX0.2;  //"DBI_QT_1".ZST.FEHLER
      JC    nexQ;
      L     %DBD24;  //"DBI_QT_1".ZST.Verweil
      +     1;
      T     %DBD24;  //"DBI_QT_1".ZST.Verweil
      AN    %DBX50.0;  //"DBI_QT_1".OUT.VOR
      AN    %DBX50.1;  //"DBI_QT_1".OUT.RUECK
      JC    nexQ;
      L     %DBD16;  //"DBI_QT_1".ZST.Dauer
      +     DINT#1;
      T     %DBD16;  //"DBI_QT_1".ZST.Dauer

nexQ: L     #Count;
      L     1;
      -I;
      JC    retQ;

wtr:  A     "DB_ANLAGE".config.Anl_getaktet;
      JC    GO;

      L     "DB_Panel_OVERVIEW".Systime;
      +     DINT#1;
      T     "DB_Panel_OVERVIEW".Systime;

      AN    "DB_ANLAGE".BA.Automat_ein;
      JC    GO;

      L     "DB_Panel_OVERVIEW".Taktzeit;
      L     1;
      +D;
      T     "DB_Panel_OVERVIEW".Taktzeit;

      L     "DB_Panel_OVERVIEW".Takt_Ware;
      L     1;
      +D;
      T     "DB_Panel_OVERVIEW".Takt_Ware;

GO:   L     "DB_ANLAGE".config.ANZ_Pos;  //Anzahl der max. abzuarbeitenden Positionen
retP: T     #anzahl;  //Prüfen ob alle Pos. abgearbeitet
      L     0;
      <=I;
      BEC;

      L     #anzahl;
      L     "DB_POS".LENG;  //Adressierung einer Position
      *I;  //und einlesen der Expozeit
      L     "DB_POS".Offset;
      +I;
      SLD   3;
      LAR1;

      OPN   "DB_POS";
      L     DBB [AR1, P#35.0];  //Ist Ware auf dieser Position?
      T     #X_DB;
      L     0;
      >I;
      JC    verw;
      T     DBD [AR1, P#76.0];
      T     DBD [AR1, P#72.0];
      T     DBW [AR1, P#70.0];  //Rest-Takte

      L     DBW [AR1, P#98.0];  //"DB_POS".POS[0].Leerzeit
      +     1;
      L     0;  //Überlauf
      <I;
      JC    DecP;
      CAC;
      T     DBW [AR1, P#98.0];  //"DB_POS".POS[0].Leerzeit
      JU    DecP;

verw: L     DBD [AR1, P#76.0];  //Verweilzeit um 1 inkrementieren
      L     16#0000_0001;
      +D;
      T     DBD [AR1, P#76.0];

      L     0;  //Leerstandzeit reset
      T     DBW [AR1, P#98.0];  //"DB_POS".POS[0].Leerzeit

goEx: L     DBD [AR1, P#44.0];  //Soll_Expozeit
      L     DBD [AR1, P#88.0];  //WaitTime
      +D;
      L     DBD [AR1, P#76.0];  //Verweilzeit
      -D;
      JPZ   expo;

      L     #X_DB;  //SaveTime am WT zählen
      L     100;
      +I;
      T     #X_DB;
      OPN   DB [#X_DB];
      L     %DBD50;
      L     0;
      <=D;
      JC    KorT;
      CAC;
      L     1;
      -D;
KorT: T     %DBD50;

      L     0;
expo: OPN   "DB_POS";
      T     DBD [AR1, P#72.0];  //Ist_Expozeit
DecP: L     #anzahl;
      L     1;
      -I;
      JU    retP;
END_FUNCTION

FUNCTION "FC_FW_Auftrag_Befehl" : Void   // FC187, LAD
{ S7_Optimized_Access := 'TRUE' }
// stored: AutoNumber false, SetENOAutomatically false
   VAR_INPUT
      inQuelle : Int;
      inZiel : Int;
   END_VAR
   VAR_OUTPUT
      Befehl_ok : Bool;
      outQuelle : Int;
      outZiel : Int;
   END_VAR
   VAR_TEMP
      kl_Ziel : Int;
      gr_Ziel : Int;
      Befehl : DWord;
      vor : Bool;
      erlaubt : Bool;
      chk_on : Bool;
      leer : Bool;
   END_VAR
BEGIN

REGION Network 1 (SCL)
   #Befehl_ok := FALSE;
   #outQuelle := 0;
   #outZiel := 0;

   #vor := #inZiel >= #inQuelle;
   #leer := #inZiel = 0;

   IF #leer THEN
       #kl_Ziel := #inZiel;
       #gr_Ziel := #inZiel;
   ELSIF #vor THEN
       #kl_Ziel := #inQuelle;
       #gr_Ziel := #inZiel;
   ELSE
       #kl_Ziel := #inZiel;
       #gr_Ziel := #inQuelle;
   END_IF;

   #chk_on := FALSE;// ("DB_POS".POS[#inQuelle].WT_DB <> 0) AND "DB_POS".POS[#inQuelle].fertig;

   IF NOT #leer THEN
       IF ("DB_POS".POS[#inQuelle].next_WT = 0) OR NOT "DB_POS".POS[#inQuelle].belegt THEN
           RETURN;
       END_IF;

       IF "DB_POS".POS[#inQuelle].Quelle OR "DB_POS".POS[#inQuelle].Sperre_out OR "DB_POS".POS[#inQuelle].notFG_out THEN
           RETURN;
       END_IF;

       IF ("DB_POS".POS[#inZiel].next_WT <> "DB_POS".POS[#inQuelle].next_WT) THEN
           IF ("DB_POS".POS[#inZiel].next_WT <> 0) OR "DB_POS".POS[#inZiel].belegt THEN
               RETURN;
           END_IF;
       END_IF;

       IF "DB_POS".POS[#inZiel].Ziel OR "DB_POS".POS[#inZiel].Sperre_in OR "DB_POS".POS[#inZiel].notFG_in THEN
           RETURN;
       END_IF;

   END_IF;

   "FC_FW_Befehl_ok"(FW_Nr:=1,
                     kl_Z:=#kl_Ziel,
                     Gr_Z:=#gr_Ziel,
                     QT_Check:=TRUE,
                     Ablassen:=FALSE,
                     vor:=#vor,
                     chk_on:=#chk_on,
                     erlaubt=>#erlaubt);

   IF NOT #erlaubt OR NOT "DI_FW_1".ZST.BEREIT THEN
       RETURN;
   END_IF;

   IF #leer THEN
       #Befehl := dw#16#F0010000;
   ELSE
       #Befehl := dw#16#F0030000;
   END_IF;

   #Befehl := #Befehl OR SHL_INT(IN:=#inQuelle,N:=8) OR #inZiel;
   "DI_FW_1".ZST.BEFEHL := #Befehl;

   #Befehl_ok := TRUE;
   #outQuelle := #inQuelle;
   #outZiel := #inZiel;
END_REGION
END_FUNCTION

FUNCTION "FC_FW_Auftrag_Parken" : Void   // FC186, LAD
{ S7_Optimized_Access := 'TRUE' }
// stored: AutoNumber false, SetENOAutomatically false
   VAR_OUTPUT
      nextStep : Bool;
      startStep : Bool;
   END_VAR
   VAR_IN_OUT
      Quelle : Int;
      Ziel : Int;
      Positionen : Array[1..30] of "UDT_Auftrag_Pos";
   END_VAR
   VAR_TEMP
      Befehl_ok : Bool;
   END_VAR
BEGIN

REGION Network 1 (SCL)
   IF (#Quelle <> 0) AND (#Ziel <> 0) THEN
       #nextStep := #Positionen[#Quelle].Sperre;
       #startStep := NOT #nextStep;
       #Quelle := 0;
       #Ziel := 0;
       RETURN;
   END_IF;

   #Quelle := 0;
   #Ziel := 0;
   #nextStep := FALSE;
   #startStep := FALSE;
END_REGION

REGION Network 2 (SCL): Transportwagen schieben
   //CM01
   IF ("DI_FW_1".ZST.POSITION_li <= 6) THEN
       "FC_FW_Auftrag_Befehl"(inQuelle := 7,
                              inZiel := 0,
                              Befehl_ok => #Befehl_ok,
                              outQuelle => #Quelle,
                              outZiel => #Ziel);

       #nextStep := NOT #Befehl_ok;
       RETURN;
   END_IF;

   //CM02
   IF ("DI_FW_1".ZST.POSITION_li >= 13) AND ("DI_FW_1".ZST.POSITION_li <= 18) THEN
       "FC_FW_Auftrag_Befehl"(inQuelle := 11,
                              inZiel := 0,
                              Befehl_ok => #Befehl_ok,
                              outQuelle => #Quelle,
                              outZiel => #Ziel);

       #nextStep := NOT #Befehl_ok;
       RETURN;
   END_IF;

   //WR02
   IF ("DI_FW_1".ZST.POSITION_li >= 25) THEN
       "FC_FW_Auftrag_Befehl"(inQuelle := 23,
                              inZiel := 0,
                              Befehl_ok => #Befehl_ok,
                              outQuelle => #Quelle,
                              outZiel => #Ziel);

       #nextStep := NOT #Befehl_ok;
       RETURN;
   END_IF;

   //?
   #nextStep := TRUE;
END_REGION
END_FUNCTION

FUNCTION "FC_FW_Auftrag_Step1_KB" : Void   // FC1081, LAD
TITLE = Schritt CM01/CMD02 -> CM03/CM04
{ S7_Optimized_Access := 'TRUE' }
// Ältesten Warenträger in CM01/CM02 suchen und nach CM03 bzw. CM04 transportieren
// stored: AutoNumber false, SetENOAutomatically false
   VAR_INPUT
      Frg_Schritt : Bool;
   END_VAR
   VAR_OUTPUT
      nextStep : Bool;
      startStep : Bool;
      parkStep : Bool;
   END_VAR
   VAR_IN_OUT
      Quelle : Int;
      Ziel : Int;
      Positionen : Array[1..30] of "UDT_Auftrag_Pos";
   END_VAR
   VAR_TEMP
      Sperre_Kurz_li_CM03 : Bool;
      Sperre_Kurz_re_CM03 : Bool;
      Sperre_Lang_CM03 : Bool;
      Sperre_Kurz_li_CM04 : Bool;
      Sperre_Kurz_re_CM04 : Bool;
      Sperre_Lang_CM04 : Bool;
      Vorzug : Bool;
      Befehl_ok : Bool;
      tmpQuelle : Int;
      Oldest : Real;
   END_VAR
BEGIN

REGION Network 1 (SCL): Initialisieren
   IF (#Quelle <> 0) AND (#Ziel <> 0) THEN
       #nextStep := #Positionen[#Quelle].Sperre;
       #startStep := NOT #nextStep;
       #Quelle := 0;
       #Ziel := 0;
       RETURN;
   END_IF;

   #Quelle := 0;
   #Ziel := 0;
   #nextStep := FALSE;
   #startStep := FALSE;

   IF NOT #Frg_Schritt THEN
       #nextStep := TRUE;
       RETURN;
   END_IF;
END_REGION

REGION Network 2 (SCL): Positionen sperren
   //Groß links nicht möglich
   #Positionen[3].CheckSperre := #Positionen[9].Sperre;
   #Positionen[15].CheckSperre := #Positionen[21].Sperre;

   //Groß rechts nicht möglich
   #Positionen[4].CheckSperre := #Positionen[10].Sperre;
   #Positionen[16].CheckSperre := #Positionen[22].Sperre;

   //kein Platz für Kurz links in CM03
   #Sperre_Kurz_li_CM03 := #Positionen[7].Sperre AND #Positionen[11].Sperre;

   //kein Platz für Kurz rechts in CM03
   #Sperre_Kurz_re_CM03 := #Positionen[8].Sperre AND #Positionen[12].Sperre;

   //kein Platz für Lang in CM03
   #Sperre_Lang_CM03 := (#Positionen[7].Sperre OR #Positionen[8].Sperre) AND (#Positionen[11].Sperre OR #Positionen[12].Sperre);

   //kein Platz für Kurz links in CM04
   #Sperre_Kurz_li_CM04 := #Positionen[19].Sperre AND #Positionen[23].Sperre;

   //kein Platz für Kurz rechts in CM04
   #Sperre_Kurz_re_CM04 := #Positionen[20].Sperre AND #Positionen[24].Sperre;

   //kein Platz für Lang in CM04
   #Sperre_Lang_CM04 := (#Positionen[19].Sperre OR #Positionen[20].Sperre) AND (#Positionen[23].Sperre OR #Positionen[24].Sperre);


   //Lang in P1 oder
   //kein Platz auf rechter Seite
   //-> P2 sperren
   #Positionen[2].CheckSperre := #Sperre_Kurz_re_CM03 OR (#Positionen[1].Wt_Typ = "WT_Typ_LS");

   //Lang in P1 und kein Platz für Lang oder
   //kein Platz auf linker Seite
   //-> P1 sperren
   #Positionen[1].CheckSperre := #Sperre_Kurz_li_CM03 OR ((#Positionen[1].Wt_Typ = "WT_Typ_LS") AND #Sperre_Lang_CM03);

   //Lang in P5 oder
   //kein Platz auf rechter Seite
   //-> P6 sperren
   #Positionen[6].CheckSperre := #Sperre_Kurz_re_CM03 OR (#Positionen[5].Wt_Typ = "WT_Typ_LS");

   //Lang in P5 und kein Platz für Lang oder
   //kein Platz auf linker Seite
   //-> P5 sperren
   #Positionen[5].CheckSperre := #Sperre_Kurz_li_CM03 OR ((#Positionen[5].Wt_Typ = "WT_Typ_LS") AND #Sperre_Lang_CM03);

   //Lang in P13 oder
   //kein Platz auf rechter Seite
   //-> P14 sperren
   #Positionen[14].CheckSperre := #Sperre_Kurz_re_CM04 OR (#Positionen[13].Wt_Typ = "WT_Typ_LS");

   //Lang in P13 und kein Platz für Lang oder
   //kein Platz auf linker Seite
   //-> P13 sperren
   #Positionen[13].CheckSperre := #Sperre_Kurz_li_CM04 OR ((#Positionen[13].Wt_Typ = "WT_Typ_LS") AND #Sperre_Lang_CM04);

   //Lang in P17 oder
   //kein Platz auf rechter Seite
   //-> P18 sperren
   #Positionen[18].CheckSperre := #Sperre_Kurz_re_CM04 OR (#Positionen[17].Wt_Typ = "WT_Typ_LS");

   //Lang in P17 und kein Platz für Lang oder
   //kein Platz auf linker Seite
   //-> P17 sperren
   #Positionen[17].CheckSperre := #Sperre_Kurz_li_CM04 OR ((#Positionen[17].Wt_Typ = "WT_Typ_LS") AND #Sperre_Lang_CM04);
END_REGION

REGION Network 3 (SCL): Ältesten WT suchen
   //
   #Oldest := 0;
   #tmpQuelle := 0;

   //CM01
   "FC_FW_Auftrag_Suche"(Pos1 := 1,
                         Pos2 := 6,
                         Positionen := #Positionen,
                         Quelle := #tmpQuelle,
                         Oldest := #Oldest);

   //CM02
   "FC_FW_Auftrag_Suche"(Pos1 := 13,
                         Pos2 := 18,
                         Positionen := #Positionen,
                         Quelle := #tmpQuelle,
                         Oldest := #Oldest);
END_REGION

REGION Network 4 (SCL): Auswertung
   IF #tmpQuelle = 0 THEN
       //kein WT
       #nextStep := TRUE;
       RETURN;
   END_IF;

   IF ("DI_FW_1".ZST.POSITION_li <= 6) AND (#tmpQuelle <= 6) THEN
       //schieben wenn über Quelle CM01
       "FC_FW_Auftrag_Befehl"(inQuelle := 7,
                              inZiel := 0,
                              Befehl_ok => #Befehl_ok,
                              outQuelle => #Quelle,
                              outZiel => #Ziel);

       #nextStep := NOT #Befehl_ok;
       RETURN;
   END_IF;

   IF ("DI_FW_1".ZST.POSITION_li >= 13) AND ("DI_FW_1".ZST.POSITION_li <= 18) AND (#tmpQuelle >= 13) THEN
       //schieben wenn über Quelle CM02
       "FC_FW_Auftrag_Befehl"(inQuelle := 11,
                              inZiel := 0,
                              Befehl_ok => #Befehl_ok,
                              outQuelle => #Quelle,
                              outZiel => #Ziel);

       #nextStep := NOT #Befehl_ok;
       RETURN;
   END_IF;

   IF NOT #Positionen[#tmpQuelle].Fertig THEN
       #parkStep := TRUE;
       RETURN;
   END_IF;
   // nur "161" GO  --> CM03
   IF (#tmpQuelle = 3) THEN
       //Gross links
       IF NOT #Positionen[9].Sperre THEN
           "FC_FW_Auftrag_Befehl"(inQuelle := #tmpQuelle,
                                  inZiel := 9,
                                  Befehl_ok => #Befehl_ok,
                                  outQuelle => #Quelle,
                                  outZiel => #Ziel);

           #nextStep := NOT #Befehl_ok;
       ELSE
           #nextStep := TRUE;
       END_IF;
       RETURN;
   END_IF;

   IF (#tmpQuelle = 4) OR (#tmpQuelle = 16) THEN
       //Gross rechts
       IF NOT #Positionen[10].Sperre THEN
           "FC_FW_Auftrag_Befehl"(inQuelle := #tmpQuelle,
                                  inZiel := 10,
                                  Befehl_ok => #Befehl_ok,
                                  outQuelle => #Quelle,
                                  outZiel => #Ziel);

           #nextStep := NOT #Befehl_ok;
       ELSE
           #nextStep := TRUE;
       END_IF;
       RETURN;
   END_IF;

   IF (#Positionen[#tmpQuelle].Wt_Typ = "WT_Typ_LS") AND ((#tmpQuelle = 1) OR (#tmpQuelle = 5)) THEN
       //Lang "161"
       IF NOT #Positionen[7].Sperre AND NOT #Positionen[8].Sperre THEN
           "FC_FW_Auftrag_Befehl"(inQuelle := #tmpQuelle,
                                  inZiel := 7,
                                  Befehl_ok => #Befehl_ok,
                                  outQuelle => #Quelle,
                                  outZiel => #Ziel);

           #nextStep := NOT #Befehl_ok;
       ELSIF NOT #Positionen[11].Sperre AND NOT #Positionen[12].Sperre THEN
           "FC_FW_Auftrag_Befehl"(inQuelle := #tmpQuelle,
                                  inZiel := 11,
                                  Befehl_ok => #Befehl_ok,
                                  outQuelle => #Quelle,
                                  outZiel => #Ziel);

           #nextStep := NOT #Befehl_ok;
       ELSE
           #nextStep := TRUE;
       END_IF;
       RETURN;
   END_IF;

   IF (#Positionen[#tmpQuelle].Wt_Typ = "WT_Typ_LS") AND ((#tmpQuelle = 13) OR (#tmpQuelle = 17)) THEN
       //Lang "151"
       IF NOT #Positionen[19].Sperre AND NOT #Positionen[20].Sperre THEN
           "FC_FW_Auftrag_Befehl"(inQuelle := #tmpQuelle,
                                  inZiel := 19,
                                  Befehl_ok => #Befehl_ok,
                                  outQuelle => #Quelle,
                                  outZiel => #Ziel);

           #nextStep := NOT #Befehl_ok;
       ELSIF NOT #Positionen[23].Sperre AND NOT #Positionen[24].Sperre THEN
           "FC_FW_Auftrag_Befehl"(inQuelle := #tmpQuelle,
                                  inZiel := 23,
                                  Befehl_ok => #Befehl_ok,
                                  outQuelle => #Quelle,
                                  outZiel => #Ziel);

           #nextStep := NOT #Befehl_ok;
       ELSE
           #nextStep := TRUE;
       END_IF;
       RETURN;
   END_IF;

   IF (#tmpQuelle = 1) OR (#tmpQuelle = 5)  THEN
       //Kurz links "161"
       #Vorzug := NOT #Positionen[7].Sperre AND NOT #Positionen[8].Sperre AND NOT #Positionen[11].Sperre AND #Positionen[12].Sperre;

       IF NOT #Positionen[7].Sperre AND NOT #Vorzug THEN
           "FC_FW_Auftrag_Befehl"(inQuelle := #tmpQuelle,
                                  inZiel := 7,
                                  Befehl_ok => #Befehl_ok,
                                  outQuelle => #Quelle,
                                  outZiel => #Ziel);

           #nextStep := NOT #Befehl_ok;
       ELSIF NOT #Positionen[11].Sperre THEN
           "FC_FW_Auftrag_Befehl"(inQuelle := #tmpQuelle,
                                  inZiel := 11,
                                  Befehl_ok => #Befehl_ok,
                                  outQuelle => #Quelle,
                                  outZiel => #Ziel);

           #nextStep := NOT #Befehl_ok;
       ELSE
           #nextStep := TRUE;
       END_IF;
       RETURN;
   END_IF;

   IF (#tmpQuelle = 13) OR (#tmpQuelle = 17) THEN
       //Kurz links "151"
       #Vorzug := NOT #Positionen[19].Sperre AND NOT #Positionen[20].Sperre AND NOT #Positionen[23].Sperre AND #Positionen[24].Sperre;

       IF NOT #Positionen[19].Sperre AND NOT #Vorzug THEN
           "FC_FW_Auftrag_Befehl"(inQuelle := #tmpQuelle,
                                  inZiel := 19,
                                  Befehl_ok => #Befehl_ok,
                                  outQuelle => #Quelle,
                                  outZiel => #Ziel);

           #nextStep := NOT #Befehl_ok;
       ELSIF NOT #Positionen[23].Sperre THEN
           "FC_FW_Auftrag_Befehl"(inQuelle := #tmpQuelle,
                                  inZiel := 23,
                                  Befehl_ok => #Befehl_ok,
                                  outQuelle => #Quelle,
                                  outZiel => #Ziel);

           #nextStep := NOT #Befehl_ok;
       ELSE
           #nextStep := TRUE;
       END_IF;
       RETURN;
   END_IF;


   IF (#tmpQuelle = 2) OR (#tmpQuelle = 6) THEN
       //Kurz rechts "161"
       #Vorzug := NOT #Positionen[7].Sperre AND NOT #Positionen[8].Sperre AND #Positionen[11].Sperre AND NOT #Positionen[12].Sperre;

       IF NOT #Positionen[8].Sperre AND NOT #Vorzug THEN
           "FC_FW_Auftrag_Befehl"(inQuelle := #tmpQuelle,
                                  inZiel := 8,
                                  Befehl_ok => #Befehl_ok,
                                  outQuelle => #Quelle,
                                  outZiel => #Ziel);

           #nextStep := NOT #Befehl_ok;
       ELSIF NOT #Positionen[12].Sperre THEN
           "FC_FW_Auftrag_Befehl"(inQuelle := #tmpQuelle,
                                  inZiel := 12,
                                  Befehl_ok => #Befehl_ok,
                                  outQuelle => #Quelle,
                                  outZiel => #Ziel);

           #nextStep := NOT #Befehl_ok;
       ELSE
           #nextStep := TRUE;
       END_IF;
       RETURN;
   END_IF;


   IF (#tmpQuelle = 14) OR (#tmpQuelle = 18) THEN
       //Kurz rechts "151"
       #Vorzug := NOT #Positionen[19].Sperre AND NOT #Positionen[20].Sperre AND #Positionen[23].Sperre AND NOT #Positionen[24].Sperre;

